LIN {X 0,Y 697.219,Z 878.166,A -85,B 0,C 180,E1 4075.669,E2 4075.669} C_VEL
LIN {X 0,Y 690.417,Z 859.31,A -85,B 0,C 180,E1 4076.202,E2 4076.202} C_VEL
LIN {X 0,Y 690.418,Z 859.31,A -85,B 0,C 180,E1 4081.164,E2 4081.164} C_VEL
LIN {X 0,Y 690.448,Z 859.31,A -85,B 0,C 180,E1 4086.339,E2 4086.339} C_VEL
LIN {X 0,Y 690.273,Z 859.31,A -85,B 0,C 180,E1 4091.743,E2 4091.743} C_VEL
LIN {X 0,Y 690.253,Z 859.31,A -85,B 0,C 180,E1 4097.131,E2 4097.131} C_VEL
LIN {X 0,Y 690.435,Z 859.31,A -85,B 0,C 180,E1 4102.194,E2 4102.194} C_VEL
LIN {X 0,Y 690.368,Z 859.31,A -85,B 0,C 180,E1 4106.732,E2 4106.732} C_VEL
LIN {X 0,Y 690.473,Z 859.31,A -85,B 0,C 180,E1 4112.567,E2 4112.567} C_VEL
LIN {X 0,Y 690.577,Z 859.31,A -85,B 0,C 180,E1 4117.159,E2 4117.159} C_VEL
LIN {X 0,Y 690.259,Z 859.31,A -85,B 0,C 180,E1 4122.108,E2 4122.108} C_VEL
LIN {X 0,Y 690.493,Z 859.31,A -85,B 0,C 180,E1 4127.328,E2 4127.328} C_VEL
LIN {X 0,Y 690.762,Z 859.31,A -85,B 0,C 180,E1 4132.441,E2 4132.441} C_VEL
LIN {X 0,Y 690.867,Z 859.31,A -85,B 0,C 180,E1 4137.488,E2 4137.488} C_VEL
LIN {X 0,Y 690.736,Z 859.31,A -85,B 0,C 180,E1 4142.516,E2 4142.516} C_VEL
LIN {X 0,Y 690.678,Z 859.31,A -85,B 0,C 180,E1 4146.298,E2 4146.298} C_VEL
LIN {X 0,Y 690.573,Z 859.31,A -85,B 0,C 180,E1 4151.388,E2 4151.388} C_VEL
LIN {X 0,Y 690.673,Z 859.31,A -85,B 0,C 180,E1 4156.569,E2 4156.569} C_VEL
LIN {X 0,Y 690.58,Z 859.31,A -85,B 0,C 180,E1 4158.902,E2 4158.902} C_VEL
LIN {X 0,Y 689.346,Z 859.31,A -85,B 0,C 180,E1 4159.621,E2 4159.621} C_VEL
LIN {X 0,Y 682.724,Z 859.31,A -85,B 0,C 180,E1 4161.574,E2 4161.574} C_VEL
LIN {X 0,Y 682.632,Z 859.31,A -85,B 0,C 180,E1 4161.759,E2 4161.759} C_VEL
LIN {X 0,Y 682.573,Z 859.31,A -85,B 0,C 180,E1 4166.353,E2 4166.353} C_VEL
LIN {X 0,Y 682.473,Z 859.31,A -85,B 0,C 180,E1 4170.701,E2 4170.701} C_VEL
LIN {X 0,Y 682.429,Z 859.31,A -85,B 0,C 180,E1 4175.253,E2 4175.253} C_VEL
LIN {X 0,Y 682.32,Z 859.31,A -85,B 0,C 180,E1 4180.082,E2 4180.082} C_VEL
LIN {X 0,Y 682.342,Z 859.31,A -85,B 0,C 180,E1 4185.273,E2 4185.273} C_VEL
LIN {X 0,Y 682.313,Z 859.31,A -85,B 0,C 180,E1 4189.906,E2 4189.906} C_VEL
LIN {X 0,Y 682.596,Z 859.31,A -85,B 0,C 180,E1 4195.202,E2 4195.202} C_VEL
LIN {X 0,Y 682.589,Z 859.31,A -85,B 0,C 180,E1 4196.549,E2 4196.549} C_VEL
LIN {X 0,Y 694.66,Z 886.241,A -85,B 0,C 180,E1 4197.535,E2 4197.535} C_VEL
LIN {X 0,Y 694.161,Z 942.115,A -85,B 0,C 180,E1 4198.336,E2 4198.336} C_VEL
LIN {X 0,Y 692.613,Z 987.576,A -85,B 0,C 180,E1 4199.516,E2 4199.516} C_VEL
LIN {X 0,Y 690.947,Z 1031.433,A -85,B 0,C 180,E1 4201.237,E2 4201.237} C_VEL
LIN {X 0,Y 689.086,Z 1070.916,A -85,B 0,C 180,E1 4203.334,E2 4203.334} C_VEL
LIN {X 0,Y 687.326,Z 1107.752,A -85,B 0,C 180,E1 4205.869,E2 4205.869} C_VEL
LIN {X 0,Y 685.7,Z 1142.826,A -85,B 0,C 180,E1 4208.975,E2 4208.975} C_VEL
LIN {X 0,Y 684.392,Z 1172.804,A -85,B 0,C 180,E1 4212.399,E2 4212.399} C_VEL
LIN {X 0,Y 683.648,Z 1196.132,A -85,B 0,C 180,E1 4215.888,E2 4215.888} C_VEL
LIN {X 0,Y 683.29,Z 1213.836,A -85,B 0,C 180,E1 4219.458,E2 4219.458} C_VEL
LIN {X 0,Y 683.115,Z 1226.068,A -85,B 0,C 180,E1 4222.992,E2 4222.992} C_VEL
LIN {X 0,Y 682.989,Z 1233.087,A -85,B 0,C 180,E1 4226.507,E2 4226.507} C_VEL
LIN {X 0,Y 683.008,Z 1235.5,A -85,B 0,C 180,E1 4230,E2 4230} C_VEL
LIN {X 0,Y 683.027,Z 1232.652,A -85,B 0,C 180,E1 4233.816,E2 4233.816} C_VEL
LIN {X 0,Y 683.081,Z 1226.069,A -85,B 0,C 180,E1 4237.008,E2 4237.008} C_VEL
LIN {X 0,Y 683.26,Z 1213.838,A -85,B 0,C 180,E1 4240.542,E2 4240.542} C_VEL
LIN {X 0,Y 683.653,Z 1196.132,A -85,B 0,C 180,E1 4244.111,E2 4244.111} C_VEL
LIN {X 0,Y 684.375,Z 1172.883,A -85,B 0,C 180,E1 4247.591,E2 4247.591} C_VEL
LIN {X 0,Y 685.586,Z 1144.349,A -85,B 0,C 180,E1 4250.869,E2 4250.869} C_VEL
LIN {X 0,Y 687.099,Z 1111.989,A -85,B 0,C 180,E1 4253.791,E2 4253.791} C_VEL
LIN {X 0,Y 688.909,Z 1076.012,A -85,B 0,C 180,E1 4256.35,E2 4256.35} C_VEL
LIN {X 0,Y 690.795,Z 1036.511,A -85,B 0,C 180,E1 4258.528,E2 4258.528} C_VEL
LIN {X 0,Y 692.579,Z 992.801,A -85,B 0,C 180,E1 4260.303,E2 4260.303} C_VEL
LIN {X 0,Y 693.916,Z 952.719,A -85,B 0,C 180,E1 4261.43,E2 4261.43} C_VEL
LIN {X 0,Y 694.73,Z 909.018,A -85,B 0,C 180,E1 4262.187,E2 4262.187} C_VEL
LIN {X 0,Y 694.325,Z 885.263,A -85,B 0,C 180,E1 4262.495,E2 4262.495} C_VEL
LIN {X 0,Y 682.567,Z 859.31,A -85,B 0,C 180,E1 4263.452,E2 4263.452} C_VEL
LIN {X 0,Y 682.392,Z 859.31,A -85,B 0,C 180,E1 4269.011,E2 4269.011} C_VEL
LIN {X 0,Y 682.579,Z 859.31,A -85,B 0,C 180,E1 4273.486,E2 4273.486} C_VEL
LIN {X 0,Y 682.368,Z 859.31,A -85,B 0,C 180,E1 4279.027,E2 4279.027} C_VEL
LIN {X 0,Y 682.363,Z 859.31,A -85,B 0,C 180,E1 4283.17,E2 4283.17} C_VEL
LIN {X 0,Y 682.444,Z 859.31,A -85,B 0,C 180,E1 4287.806,E2 4287.806} C_VEL
LIN {X 0,Y 682.632,Z 859.31,A -85,B 0,C 180,E1 4292.612,E2 4292.612} C_VEL
LIN {X 0,Y 682.664,Z 859.31,A -85,B 0,C 180,E1 4297.835,E2 4297.835} C_VEL
LIN {X 0,Y 682.691,Z 859.31,A -85,B 0,C 180,E1 4303.232,E2 4303.232} C_VEL
LIN {X 0,Y 682.688,Z 859.31,A -85,B 0,C 180,E1 4308.478,E2 4308.478} C_VEL
LIN {X 0,Y 682.896,Z 859.31,A -85,B 0,C 180,E1 4313.63,E2 4313.63} C_VEL
LIN {X 0,Y 682.841,Z 859.31,A -85,B 0,C 180,E1 4318.727,E2 4318.727} C_VEL
LIN {X 0,Y 682.863,Z 859.31,A -85,B 0,C 180,E1 4323.075,E2 4323.075} C_VEL
LIN {X 0,Y 682.774,Z 859.31,A -85,B 0,C 180,E1 4327.648,E2 4327.648} C_VEL
LIN {X 0,Y 682.771,Z 859.31,A -85,B 0,C 180,E1 4332.817,E2 4332.817} C_VEL
LIN {X 0,Y 682.691,Z 859.31,A -85,B 0,C 180,E1 4338.097,E2 4338.097} C_VEL
LIN {X 0,Y 682.561,Z 859.31,A -85,B 0,C 180,E1 4343.545,E2 4343.545} C_VEL
LIN {X 0,Y 682.547,Z 859.31,A -85,B 0,C 180,E1 4347.779,E2 4347.779} C_VEL
LIN {X 0,Y 682.439,Z 859.31,A -85,B 0,C 180,E1 4352.462,E2 4352.462} C_VEL
LIN {X 0,Y 682.458,Z 859.31,A -85,B 0,C 180,E1 4356.935,E2 4356.935} C_VEL
LIN {X 0,Y 682.378,Z 859.31,A -85,B 0,C 180,E1 4361.757,E2 4361.757} C_VEL
LIN {X 0,Y 682.362,Z 859.31,A -85,B 0,C 180,E1 4367.104,E2 4367.104} C_VEL
LIN {X 0,Y 682.426,Z 859.31,A -85,B 0,C 180,E1 4371.558,E2 4371.558} C_VEL
LIN {X 0,Y 682.493,Z 859.31,A -85,B 0,C 180,E1 4376.285,E2 4376.285} C_VEL
LIN {X 0,Y 682.432,Z 859.31,A -85,B 0,C 180,E1 4380.759,E2 4380.759} C_VEL
LIN {X 0,Y 682.609,Z 860.101,A -85,B 0,C 180,E1 4383.414,E2 4383.414} C_VEL
LIN {X 0,Y 690.644,Z 881.208,A -85,B 0,C 180,E1 4384.012,E2 4384.012} C_VEL
LIN {X 0,Y 690.138,Z 969.054,A -85,B 0,C 180,E1 4385.079,E2 4385.079} C_VEL
LIN {X 0,Y 689.243,Z 1008.749,A -85,B 0,C 180,E1 4386.059,E2 4386.059} C_VEL
LIN {X 0,Y 687.984,Z 1047.945,A -85,B 0,C 180,E1 4387.578,E2 4387.578} C_VEL
LIN {X 0,Y 686.6,Z 1083.977,A -85,B 0,C 180,E1 4389.557,E2 4389.557} C_VEL
LIN {X 0,Y 685.347,Z 1115.624,A -85,B 0,C 180,E1 4391.886,E2 4391.886} C_VEL
LIN {X 0,Y 684.434,Z 1141.565,A -85,B 0,C 180,E1 4394.374,E2 4394.374} C_VEL
LIN {X 0,Y 683.7,Z 1165.212,A -85,B 0,C 180,E1 4397.358,E2 4397.358} C_VEL
LIN {X 0,Y 683.315,Z 1182.757,A -85,B 0,C 180,E1 4400.374,E2 4400.374} C_VEL
LIN {X 0,Y 683.103,Z 1195.738,A -85,B 0,C 180,E1 4403.632,E2 4403.632} C_VEL
LIN {X 0,Y 683.082,Z 1202.285,A -85,B 0,C 180,E1 4406.328,E2 4406.328} C_VEL
LIN {X 0,Y 683.01,Z 1205.493,A -85,B 0,C 180,E1 4410,E2 4410} C_VEL
LIN {X 0,Y 683.084,Z 1203.836,A -85,B 0,C 180,E1 4412.543,E2 4412.543} C_VEL
LIN {X 0,Y 683.168,Z 1197.388,A -85,B 0,C 180,E1 4415.728,E2 4415.728} C_VEL
LIN {X 0,Y 683.254,Z 1185.646,A -85,B 0,C 180,E1 4418.931,E2 4418.931} C_VEL
LIN {X 0,Y 683.675,Z 1167.868,A -85,B 0,C 180,E1 4422.155,E2 4422.155} C_VEL
LIN {X 0,Y 684.244,Z 1145.639,A -85,B 0,C 180,E1 4425.083,E2 4425.083} C_VEL
LIN {X 0,Y 685.221,Z 1119.372,A -85,B 0,C 180,E1 4427.702,E2 4427.702} C_VEL
LIN {X 0,Y 686.442,Z 1088.334,A -85,B 0,C 180,E1 4430.068,E2 4430.068} C_VEL
LIN {X 0,Y 687.73,Z 1053.775,A -85,B 0,C 180,E1 4432.05,E2 4432.05} C_VEL
LIN {X 0,Y 688.945,Z 1018.152,A -85,B 0,C 180,E1 4433.536,E2 4433.536} C_VEL
LIN {X 0,Y 689.856,Z 981.67,A -85,B 0,C 180,E1 4434.576,E2 4434.576} C_VEL
LIN {X 0,Y 690.349,Z 943.118,A -85,B 0,C 180,E1 4435.21,E2 4435.21} C_VEL
LIN {X 0,Y 690.062,Z 880.068,A -85,B 0,C 180,E1 4435.934,E2 4435.934} C_VEL
LIN {X 0,Y 682.529,Z 859.31,A -85,B 0,C 180,E1 4436.555,E2 4436.555} C_VEL
LIN {X 0,Y 682.492,Z 859.31,A -85,B 0,C 180,E1 4442.199,E2 4442.199} C_VEL
LIN {X 0,Y 682.491,Z 859.31,A -85,B 0,C 180,E1 4446.961,E2 4446.961} C_VEL
LIN {X 0,Y 682.387,Z 859.31,A -85,B 0,C 180,E1 4451.773,E2 4451.773} C_VEL
LIN {X 0,Y 682.353,Z 859.31,A -85,B 0,C 180,E1 4457.124,E2 4457.124} C_VEL
LIN {X 0,Y 682.4,Z 859.31,A -85,B 0,C 180,E1 4461.57,E2 4461.57} C_VEL
LIN {X 0,Y 682.466,Z 859.31,A -85,B 0,C 180,E1 4466.296,E2 4466.296} C_VEL
LIN {X 0,Y 682.56,Z 859.31,A -85,B 0,C 180,E1 4472.222,E2 4472.222} C_VEL
LIN {X 0,Y 682.612,Z 859.31,A -85,B 0,C 180,E1 4476.457,E2 4476.457} C_VEL
LIN {X 0,Y 682.546,Z 859.31,A -85,B 0,C 180,E1 4480.556,E2 4480.556} C_VEL
LIN {X 0,Y 682.564,Z 859.31,A -85,B 0,C 180,E1 4485.871,E2 4485.871} C_VEL
LIN {X 0,Y 682.778,Z 859.31,A -85,B 0,C 180,E1 4491.067,E2 4491.067} C_VEL
LIN {X 0,Y 682.942,Z 859.31,A -85,B 0,C 180,E1 4496.186,E2 4496.186} C_VEL
LIN {X 0,Y 683.061,Z 859.31,A -85,B 0,C 180,E1 4501.273,E2 4501.273} C_VEL
LIN {X 0,Y 682.784,Z 859.31,A -85,B 0,C 180,E1 4506.371,E2 4506.371} C_VEL
LIN {X 0,Y 682.666,Z 859.31,A -85,B 0,C 180,E1 4511.522,E2 4511.522} C_VEL
LIN {X 0,Y 682.744,Z 859.31,A -85,B 0,C 180,E1 4516.767,E2 4516.767} C_VEL
LIN {X 0,Y 682.632,Z 859.31,A -85,B 0,C 180,E1 4521.759,E2 4521.759} C_VEL
LIN {X 0,Y 681.37,Z 859.31,A -85,B 0,C 180,E1 4522.485,E2 4522.485} C_VEL
LIN {X 0,Y 674.718,Z 859.31,A -85,B 0,C 180,E1 4524.458,E2 4524.458} C_VEL
LIN {X 0,Y 674.625,Z 859.31,A -85,B 0,C 180,E1 4524.645,E2 4524.645} C_VEL
LIN {X 0,Y 674.577,Z 859.31,A -85,B 0,C 180,E1 4529.609,E2 4529.609} C_VEL
LIN {X 0,Y 674.523,Z 859.31,A -85,B 0,C 180,E1 4534.159,E2 4534.159} C_VEL
LIN {X 0,Y 674.482,Z 859.31,A -85,B 0,C 180,E1 4538.97,E2 4538.97} C_VEL
LIN {X 0,Y 674.429,Z 859.31,A -85,B 0,C 180,E1 4544.135,E2 4544.135} C_VEL
LIN {X 0,Y 674.436,Z 859.31,A -85,B 0,C 180,E1 4549.794,E2 4549.794} C_VEL
LIN {X 0,Y 674.626,Z 859.31,A -85,B 0,C 180,E1 4554.268,E2 4554.268} C_VEL
LIN {X 0,Y 674.719,Z 860.083,A -85,B 0,C 180,E1 4556.128,E2 4556.128} C_VEL
LIN {X 0,Y 688.177,Z 890.762,A -85,B 0,C 180,E1 4557.246,E2 4557.246} C_VEL
LIN {X 0,Y 687.372,Z 943.616,A -85,B 0,C 180,E1 4558.022,E2 4558.022} C_VEL
LIN {X 0,Y 685.688,Z 989.724,A -85,B 0,C 180,E1 4559.246,E2 4559.246} C_VEL
LIN {X 0,Y 683.712,Z 1034.768,A -85,B 0,C 180,E1 4561.064,E2 4561.064} C_VEL
LIN {X 0,Y 681.56,Z 1076.167,A -85,B 0,C 180,E1 4563.354,E2 4563.354} C_VEL
LIN {X 0,Y 679.627,Z 1112.596,A -85,B 0,C 180,E1 4565.982,E2 4565.982} C_VEL
LIN {X 0,Y 678.016,Z 1144.493,A -85,B 0,C 180,E1 4568.902,E2 4568.902} C_VEL
LIN {X 0,Y 676.631,Z 1173.438,A -85,B 0,C 180,E1 4572.278,E2 4572.278} C_VEL
LIN {X 0,Y 675.848,Z 1196.131,A -85,B 0,C 180,E1 4575.722,E2 4575.722} C_VEL
LIN {X 0,Y 675.428,Z 1213.837,A -85,B 0,C 180,E1 4579.334,E2 4579.334} C_VEL
LIN {X 0,Y 675.218,Z 1226.068,A -85,B 0,C 180,E1 4582.91,E2 4582.91} C_VEL
LIN {X 0,Y 675.118,Z 1232.65,A -85,B 0,C 180,E1 4586.139,E2 4586.139} C_VEL
LIN {X 0,Y 675.137,Z 1235.5,A -85,B 0,C 180,E1 4590,E2 4590} C_VEL
LIN {X 0,Y 675.128,Z 1232.651,A -85,B 0,C 180,E1 4593.861,E2 4593.861} C_VEL
LIN {X 0,Y 675.18,Z 1226.069,A -85,B 0,C 180,E1 4597.09,E2 4597.09} C_VEL
LIN {X 0,Y 675.392,Z 1213.839,A -85,B 0,C 180,E1 4600.666,E2 4600.666} C_VEL
LIN {X 0,Y 675.851,Z 1196.13,A -85,B 0,C 180,E1 4604.278,E2 4604.278} C_VEL
LIN {X 0,Y 676.713,Z 1171.539,A -85,B 0,C 180,E1 4607.974,E2 4607.974} C_VEL
LIN {X 0,Y 678.114,Z 1141.776,A -85,B 0,C 180,E1 4611.384,E2 4611.384} C_VEL
LIN {X 0,Y 679.994,Z 1105.755,A -85,B 0,C 180,E1 4614.571,E2 4614.571} C_VEL
LIN {X 0,Y 682.155,Z 1066.242,A -85,B 0,C 180,E1 4617.259,E2 4617.259} C_VEL
LIN {X 0,Y 684.237,Z 1024.252,A -85,B 0,C 180,E1 4619.415,E2 4619.415} C_VEL
LIN {X 0,Y 686.078,Z 981.213,A -85,B 0,C 180,E1 4621.016,E2 4621.016} C_VEL
LIN {X 0,Y 687.436,Z 937.981,A -85,B 0,C 180,E1 4622.093,E2 4622.093} C_VEL
LIN {X 0,Y 687.755,Z 888.134,A -85,B 0,C 180,E1 4622.809,E2 4622.809} C_VEL
LIN {X 0,Y 674.633,Z 859.31,A -85,B 0,C 180,E1 4623.915,E2 4623.915} C_VEL
LIN {X 0,Y 674.513,Z 859.31,A -85,B 0,C 180,E1 4628.978,E2 4628.978} C_VEL
LIN {X 0,Y 674.668,Z 859.31,A -85,B 0,C 180,E1 4634.127,E2 4634.127} C_VEL
LIN {X 0,Y 674.487,Z 859.31,A -85,B 0,C 180,E1 4639.804,E2 4639.804} C_VEL
LIN {X 0,Y 674.432,Z 859.31,A -85,B 0,C 180,E1 4644.265,E2 4644.265} C_VEL
LIN {X 0,Y 674.542,Z 859.31,A -85,B 0,C 180,E1 4648.898,E2 4648.898} C_VEL
LIN {X 0,Y 674.702,Z 859.31,A -85,B 0,C 180,E1 4653.941,E2 4653.941} C_VEL
LIN {X 0,Y 674.735,Z 859.31,A -85,B 0,C 180,E1 4658.945,E2 4658.945} C_VEL
LIN {X 0,Y 674.764,Z 859.31,A -85,B 0,C 180,E1 4664.369,E2 4664.369} C_VEL
LIN {X 0,Y 674.856,Z 859.31,A -85,B 0,C 180,E1 4669.653,E2 4669.653} C_VEL
LIN {X 0,Y 674.899,Z 859.31,A -85,B 0,C 180,E1 4674.847,E2 4674.847} C_VEL
LIN {X 0,Y 675.011,Z 859.31,A -85,B 0,C 180,E1 4679.998,E2 4679.998} C_VEL
LIN {X 0,Y 675.106,Z 859.31,A -85,B 0,C 180,E1 4685.148,E2 4685.148} C_VEL
LIN {X 0,Y 674.799,Z 859.31,A -85,B 0,C 180,E1 4690.344,E2 4690.344} C_VEL
LIN {X 0,Y 674.786,Z 859.31,A -85,B 0,C 180,E1 4695.627,E2 4695.627} C_VEL
LIN {X 0,Y 674.731,Z 859.31,A -85,B 0,C 180,E1 4701.051,E2 4701.051} C_VEL
LIN {X 0,Y 674.634,Z 859.31,A -85,B 0,C 180,E1 4706.684,E2 4706.684} C_VEL
LIN {X 0,Y 674.525,Z 859.31,A -85,B 0,C 180,E1 4711.389,E2 4711.389} C_VEL
LIN {X 0,Y 674.494,Z 859.31,A -85,B 0,C 180,E1 4716.025,E2 4716.025} C_VEL
LIN {X 0,Y 674.449,Z 859.31,A -85,B 0,C 180,E1 4720.643,E2 4720.643} C_VEL
LIN {X 0,Y 674.414,Z 859.31,A -85,B 0,C 180,E1 4725.952,E2 4725.952} C_VEL
LIN {X 0,Y 674.504,Z 859.31,A -85,B 0,C 180,E1 4731.022,E2 4731.022} C_VEL
LIN {X 0,Y 674.589,Z 859.31,A -85,B 0,C 180,E1 4736.187,E2 4736.187} C_VEL
LIN {X 0,Y 674.546,Z 859.31,A -85,B 0,C 180,E1 4741.853,E2 4741.853} C_VEL
LIN {X 0,Y 674.64,Z 859.31,A -85,B 0,C 180,E1 4742.96,E2 4742.96} C_VEL
LIN {X 0,Y 683.587,Z 884.911,A -85,B 0,C 180,E1 4743.766,E2 4743.766} C_VEL
LIN {X 0,Y 682.976,Z 969.021,A -85,B 0,C 180,E1 4744.799,E2 4744.799} C_VEL
LIN {X 0,Y 681.97,Z 1009.288,A -85,B 0,C 180,E1 4745.805,E2 4745.805} C_VEL
LIN {X 0,Y 680.567,Z 1048.213,A -85,B 0,C 180,E1 4747.334,E2 4747.334} C_VEL
LIN {X 0,Y 679.069,Z 1084.367,A -85,B 0,C 180,E1 4749.347,E2 4749.347} C_VEL
LIN {X 0,Y 677.747,Z 1114.646,A -85,B 0,C 180,E1 4751.591,E2 4751.591} C_VEL
LIN {X 0,Y 676.664,Z 1142.43,A -85,B 0,C 180,E1 4754.288,E2 4754.288} C_VEL
LIN {X 0,Y 675.885,Z 1165.244,A -85,B 0,C 180,E1 4757.215,E2 4757.215} C_VEL
LIN {X 0,Y 675.442,Z 1183.007,A -85,B 0,C 180,E1 4760.314,E2 4760.314} C_VEL
LIN {X 0,Y 675.214,Z 1195.736,A -85,B 0,C 180,E1 4763.558,E2 4763.558} C_VEL
LIN {X 0,Y 675.205,Z 1202.016,A -85,B 0,C 180,E1 4766.14,E2 4766.14} C_VEL
LIN {X 0,Y 675.121,Z 1205.119,A -85,B 0,C 180,E1 4768.714,E2 4768.714} C_VEL
LIN {X 0,Y 675.219,Z 1205.047,A -85,B 0,C 180,E1 4771.286,E2 4771.286} C_VEL
LIN {X 0,Y 675.246,Z 1200.619,A -85,B 0,C 180,E1 4774.505,E2 4774.505} C_VEL
LIN {X 0,Y 675.389,Z 1189.741,A -85,B 0,C 180,E1 4778.061,E2 4778.061} C_VEL
LIN {X 0,Y 675.739,Z 1173.885,A -85,B 0,C 180,E1 4781.316,E2 4781.316} C_VEL
LIN {X 0,Y 676.263,Z 1153.81,A -85,B 0,C 180,E1 4784.269,E2 4784.269} C_VEL
LIN {X 0,Y 677.194,Z 1128.422,A -85,B 0,C 180,E1 4787.074,E2 4787.074} C_VEL
LIN {X 0,Y 678.461,Z 1098.701,A -85,B 0,C 180,E1 4789.574,E2 4789.574} C_VEL
LIN {X 0,Y 679.837,Z 1065.972,A -85,B 0,C 180,E1 4791.664,E2 4791.664} C_VEL
LIN {X 0,Y 681.195,Z 1030.24,A -85,B 0,C 180,E1 4793.352,E2 4793.352} C_VEL
LIN {X 0,Y 682.38,Z 992.126,A -85,B 0,C 180,E1 4794.599,E2 4794.599} C_VEL
LIN {X 0,Y 683.139,Z 953.244,A -85,B 0,C 180,E1 4795.364,E2 4795.364} C_VEL
LIN {X 0,Y 682.79,Z 881.512,A -85,B 0,C 180,E1 4796.227,E2 4796.227} C_VEL
LIN {X 0,Y 674.627,Z 859.31,A -85,B 0,C 180,E1 4796.981,E2 4796.981} C_VEL
LIN {X 0,Y 674.596,Z 859.31,A -85,B 0,C 180,E1 4802.622,E2 4802.622} C_VEL
LIN {X 0,Y 674.525,Z 859.31,A -85,B 0,C 180,E1 4808.185,E2 4808.185} C_VEL
LIN {X 0,Y 674.459,Z 859.31,A -85,B 0,C 180,E1 4812.377,E2 4812.377} C_VEL
LIN {X 0,Y 674.454,Z 859.31,A -85,B 0,C 180,E1 4817.852,E2 4817.852} C_VEL
LIN {X 0,Y 674.537,Z 859.31,A -85,B 0,C 180,E1 4822.675,E2 4822.675} C_VEL
LIN {X 0,Y 674.511,Z 859.31,A -85,B 0,C 180,E1 4827.385,E2 4827.385} C_VEL
LIN {X 0,Y 674.595,Z 859.31,A -85,B 0,C 180,E1 4831.865,E2 4831.865} C_VEL
LIN {X 0,Y 674.674,Z 859.31,A -85,B 0,C 180,E1 4837.05,E2 4837.05} C_VEL
LIN {X 0,Y 674.466,Z 859.31,A -85,B 0,C 180,E1 4841.674,E2 4841.674} C_VEL
LIN {X 0,Y 674.654,Z 859.31,A -85,B 0,C 180,E1 4847.026,E2 4847.026} C_VEL
LIN {X 0,Y 674.941,Z 859.31,A -85,B 0,C 180,E1 4852.262,E2 4852.262} C_VEL
LIN {X 0,Y 675.075,Z 859.31,A -85,B 0,C 180,E1 4857.429,E2 4857.429} C_VEL
LIN {X 0,Y 674.956,Z 859.31,A -85,B 0,C 180,E1 4862.575,E2 4862.575} C_VEL
LIN {X 0,Y 674.874,Z 859.31,A -85,B 0,C 180,E1 4866.446,E2 4866.446} C_VEL
LIN {X 0,Y 674.788,Z 859.31,A -85,B 0,C 180,E1 4870.348,E2 4870.348} C_VEL
LIN {X 0,Y 674.799,Z 859.31,A -85,B 0,C 180,E1 4875.63,E2 4875.63} C_VEL
LIN {X 0,Y 674.785,Z 859.31,A -85,B 0,C 180,E1 4881.053,E2 4881.053} C_VEL
LIN {X 0,Y 674.625,Z 859.31,A -85,B 0,C 180,E1 4884.645,E2 4884.645} C_VEL
LIN {X 0,Y 670.662,Z 859.31,A -85,B 0,C 180,E1 4886.09,E2 4886.09} C_VEL
LIN {X 0,Y 666.704,Z 859.31,A -85,B 0,C 180,E1 4887.552,E2 4887.552} C_VEL
LIN {X 0,Y 666.618,Z 859.31,A -85,B 0,C 180,E1 4893.054,E2 4893.054} C_VEL
LIN {X 0,Y 666.601,Z 859.31,A -85,B 0,C 180,E1 4897.852,E2 4897.852} C_VEL
LIN {X 0,Y 666.477,Z 859.31,A -85,B 0,C 180,E1 4903.319,E2 4903.319} C_VEL
LIN {X 0,Y 666.481,Z 859.31,A -85,B 0,C 180,E1 4908.75,E2 4908.75} C_VEL
LIN {X 0,Y 666.685,Z 859.31,A -85,B 0,C 180,E1 4913.775,E2 4913.775} C_VEL
LIN {X 0,Y 666.773,Z 859.31,A -85,B 0,C 180,E1 4915.739,E2 4915.739} C_VEL
LIN {X 0,Y 676.305,Z 880.508,A -85,B 0,C 180,E1 4916.468,E2 4916.468} C_VEL
LIN {X 0,Y 681.457,Z 891.656,A -85,B 0,C 180,E1 4916.892,E2 4916.892} C_VEL
LIN {X 0,Y 680.649,Z 943.593,A -85,B 0,C 180,E1 4917.667,E2 4917.667} C_VEL
LIN {X 0,Y 678.842,Z 989.466,A -85,B 0,C 180,E1 4918.893,E2 4918.893} C_VEL
LIN {X 0,Y 676.675,Z 1035.331,A -85,B 0,C 180,E1 4920.761,E2 4920.761} C_VEL
LIN {X 0,Y 674.296,Z 1076.831,A -85,B 0,C 180,E1 4923.087,E2 4923.087} C_VEL
LIN {X 0,Y 672.129,Z 1113.665,A -85,B 0,C 180,E1 4925.787,E2 4925.787} C_VEL
LIN {X 0,Y 670.365,Z 1145.862,A -85,B 0,C 180,E1 4928.797,E2 4928.797} C_VEL
LIN {X 0,Y 668.912,Z 1173.914,A -85,B 0,C 180,E1 4932.133,E2 4932.133} C_VEL
LIN {X 0,Y 668.036,Z 1196.13,A -85,B 0,C 180,E1 4935.551,E2 4935.551} C_VEL
LIN {X 0,Y 667.568,Z 1213.837,A -85,B 0,C 180,E1 4939.207,E2 4939.207} C_VEL
LIN {X 0,Y 667.325,Z 1226.068,A -85,B 0,C 180,E1 4942.826,E2 4942.826} C_VEL
LIN {X 0,Y 667.224,Z 1232.65,A -85,B 0,C 180,E1 4946.093,E2 4946.093} C_VEL
LIN {X 0,Y 667.237,Z 1235.5,A -85,B 0,C 180,E1 4950,E2 4950} C_VEL
LIN {X 0,Y 667.231,Z 1232.651,A -85,B 0,C 180,E1 4953.906,E2 4953.906} C_VEL
LIN {X 0,Y 667.284,Z 1226.069,A -85,B 0,C 180,E1 4957.175,E2 4957.175} C_VEL
LIN {X 0,Y 667.528,Z 1213.84,A -85,B 0,C 180,E1 4960.794,E2 4960.794} C_VEL
LIN {X 0,Y 668.037,Z 1196.129,A -85,B 0,C 180,E1 4964.448,E2 4964.448} C_VEL
LIN {X 0,Y 669.015,Z 1171.677,A -85,B 0,C 180,E1 4968.17,E2 4968.17} C_VEL
LIN {X 0,Y 670.587,Z 1141.188,A -85,B 0,C 180,E1 4971.696,E2 4971.696} C_VEL
LIN {X 0,Y 672.667,Z 1105.263,A -85,B 0,C 180,E1 4974.895,E2 4974.895} C_VEL
LIN {X 0,Y 674.957,Z 1066.239,A -85,B 0,C 180,E1 4977.574,E2 4977.574} C_VEL
LIN {X 0,Y 677.288,Z 1023.55,A -85,B 0,C 180,E1 4979.781,E2 4979.781} C_VEL
LIN {X 0,Y 679.279,Z 980.059,A -85,B 0,C 180,E1 4981.399,E2 4981.399} C_VEL
LIN {X 0,Y 680.782,Z 935.996,A -85,B 0,C 180,E1 4982.483,E2 4982.483} C_VEL
LIN {X 0,Y 680.982,Z 890.343,A -85,B 0,C 180,E1 4983.15,E2 4983.15} C_VEL
LIN {X 0,Y 666.851,Z 860.732,A -85,B 0,C 180,E1 4984.225,E2 4984.225} C_VEL
LIN {X 0,Y 666.711,Z 859.31,A -85,B 0,C 180,E1 4984.302,E2 4984.302} C_VEL
LIN {X 0,Y 666.57,Z 859.31,A -85,B 0,C 180,E1 4989.532,E2 4989.532} C_VEL
LIN {X 0,Y 666.662,Z 859.31,A -85,B 0,C 180,E1 4994.798,E2 4994.798} C_VEL
LIN {X 0,Y 666.567,Z 859.31,A -85,B 0,C 180,E1 5000.616,E2 5000.616} C_VEL
LIN {X 0,Y 666.52,Z 859.31,A -85,B 0,C 180,E1 5005.372,E2 5005.372} C_VEL
LIN {X 0,Y 666.624,Z 859.31,A -85,B 0,C 180,E1 5010.002,E2 5010.002} C_VEL
LIN {X 0,Y 666.768,Z 859.31,A -85,B 0,C 180,E1 5015.372,E2 5015.372} C_VEL
LIN {X 0,Y 666.803,Z 859.31,A -85,B 0,C 180,E1 5020.074,E2 5020.074} C_VEL
LIN {X 0,Y 666.845,Z 859.31,A -85,B 0,C 180,E1 5024.179,E2 5024.179} C_VEL
LIN {X 0,Y 666.932,Z 859.31,A -85,B 0,C 180,E1 5029.529,E2 5029.529} C_VEL
LIN {X 0,Y 667.009,Z 859.31,A -85,B 0,C 180,E1 5034.786,E2 5034.786} C_VEL
LIN {X 0,Y 667.074,Z 859.31,A -85,B 0,C 180,E1 5038.697,E2 5038.697} C_VEL
LIN {X 0,Y 667.07,Z 859.31,A -85,B 0,C 180,E1 5042.601,E2 5042.601} C_VEL
LIN {X 0,Y 666.962,Z 859.31,A -85,B 0,C 180,E1 5046.519,E2 5046.519} C_VEL
LIN {X 0,Y 666.896,Z 859.31,A -85,B 0,C 180,E1 5051.795,E2 5051.795} C_VEL
LIN {X 0,Y 666.854,Z 859.31,A -85,B 0,C 180,E1 5057.377,E2 5057.377} C_VEL
LIN {X 0,Y 666.728,Z 859.31,A -85,B 0,C 180,E1 5062.72,E2 5062.72} C_VEL
LIN {X 0,Y 666.669,Z 859.31,A -85,B 0,C 180,E1 5067.571,E2 5067.571} C_VEL
LIN {X 0,Y 666.615,Z 859.31,A -85,B 0,C 180,E1 5073.05,E2 5073.05} C_VEL
LIN {X 0,Y 666.606,Z 859.31,A -85,B 0,C 180,E1 5077.847,E2 5077.847} C_VEL
LIN {X 0,Y 666.468,Z 859.31,A -85,B 0,C 180,E1 5083.318,E2 5083.318} C_VEL
LIN {X 0,Y 666.494,Z 859.31,A -85,B 0,C 180,E1 5088.752,E2 5088.752} C_VEL
LIN {X 0,Y 666.661,Z 859.31,A -85,B 0,C 180,E1 5093.774,E2 5093.774} C_VEL
LIN {X 0,Y 666.596,Z 859.31,A -85,B 0,C 180,E1 5098.478,E2 5098.478} C_VEL
LIN {X 0,Y 666.724,Z 859.31,A -85,B 0,C 180,E1 5102.531,E2 5102.531} C_VEL
LIN {X 0,Y 676.777,Z 885.125,A -85,B 0,C 180,E1 5103.408,E2 5103.408} C_VEL
LIN {X 0,Y 675.999,Z 968.354,A -85,B 0,C 180,E1 5104.475,E2 5104.475} C_VEL
LIN {X 0,Y 674.765,Z 1007.317,A -85,B 0,C 180,E1 5105.469,E2 5105.469} C_VEL
LIN {X 0,Y 673.291,Z 1046.299,A -85,B 0,C 180,E1 5106.982,E2 5106.982} C_VEL
LIN {X 0,Y 671.684,Z 1082.811,A -85,B 0,C 180,E1 5109.004,E2 5109.004} C_VEL
LIN {X 0,Y 670.124,Z 1114.638,A -85,B 0,C 180,E1 5111.374,E2 5111.374} C_VEL
LIN {X 0,Y 668.907,Z 1142.424,A -85,B 0,C 180,E1 5114.101,E2 5114.101} C_VEL
LIN {X 0,Y 668.123,Z 1164.113,A -85,B 0,C 180,E1 5116.892,E2 5116.892} C_VEL
LIN {X 0,Y 667.624,Z 1181.463,A -85,B 0,C 180,E1 5119.869,E2 5119.869} C_VEL
LIN {X 0,Y 667.391,Z 1194.77,A -85,B 0,C 180,E1 5123.154,E2 5123.154} C_VEL
LIN {X 0,Y 667.311,Z 1202.016,A -85,B 0,C 180,E1 5126.094,E2 5126.094} C_VEL
LIN {X 0,Y 667.221,Z 1205.119,A -85,B 0,C 180,E1 5128.699,E2 5128.699} C_VEL
LIN {X 0,Y 667.317,Z 1205.047,A -85,B 0,C 180,E1 5131.301,E2 5131.301} C_VEL
LIN {X 0,Y 667.361,Z 1200.621,A -85,B 0,C 180,E1 5134.558,E2 5134.558} C_VEL
LIN {X 0,Y 667.518,Z 1189.743,A -85,B 0,C 180,E1 5138.157,E2 5138.157} C_VEL
LIN {X 0,Y 667.901,Z 1173.887,A -85,B 0,C 180,E1 5141.45,E2 5141.45} C_VEL
LIN {X 0,Y 668.474,Z 1153.813,A -85,B 0,C 180,E1 5144.439,E2 5144.439} C_VEL
LIN {X 0,Y 669.493,Z 1128.631,A -85,B 0,C 180,E1 5147.257,E2 5147.257} C_VEL
LIN {X 0,Y 670.883,Z 1098.706,A -85,B 0,C 180,E1 5149.804,E2 5149.804} C_VEL
LIN {X 0,Y 672.424,Z 1065.979,A -85,B 0,C 180,E1 5151.915,E2 5151.915} C_VEL
LIN {X 0,Y 673.932,Z 1029.418,A -85,B 0,C 180,E1 5153.654,E2 5153.654} C_VEL
LIN {X 0,Y 675.356,Z 990.18,A -85,B 0,C 180,E1 5154.939,E2 5154.939} C_VEL
LIN {X 0,Y 676.221,Z 953.656,A -85,B 0,C 180,E1 5155.681,E2 5155.681} C_VEL
LIN {X 0,Y 676.308,Z 884.254,A -85,B 0,C 180,E1 5156.536,E2 5156.536} C_VEL
LIN {X 0,Y 666.712,Z 859.31,A -85,B 0,C 180,E1 5157.403,E2 5157.403} C_VEL
LIN {X 0,Y 666.678,Z 859.31,A -85,B 0,C 180,E1 5163.059,E2 5163.059} C_VEL
LIN {X 0,Y 666.632,Z 859.31,A -85,B 0,C 180,E1 5167.86,E2 5167.86} C_VEL
LIN {X 0,Y 666.46,Z 859.31,A -85,B 0,C 180,E1 5173.336,E2 5173.336} C_VEL
LIN {X 0,Y 666.486,Z 859.31,A -85,B 0,C 180,E1 5178.767,E2 5178.767} C_VEL
LIN {X 0,Y 666.662,Z 859.31,A -85,B 0,C 180,E1 5183.788,E2 5183.788} C_VEL
LIN {X 0,Y 666.574,Z 859.31,A -85,B 0,C 180,E1 5188.488,E2 5188.488} C_VEL
LIN {X 0,Y 666.706,Z 859.31,A -85,B 0,C 180,E1 5192.973,E2 5192.973} C_VEL
LIN {X 0,Y 666.779,Z 859.31,A -85,B 0,C 180,E1 5197.282,E2 5197.282} C_VEL
LIN {X 0,Y 666.586,Z 859.31,A -85,B 0,C 180,E1 5201.45,E2 5201.45} C_VEL
LIN {X 0,Y 666.751,Z 859.31,A -85,B 0,C 180,E1 5206.869,E2 5206.869} C_VEL
LIN {X 0,Y 667.027,Z 859.31,A -85,B 0,C 180,E1 5212.17,E2 5212.17} C_VEL
LIN {X 0,Y 667.197,Z 859.31,A -85,B 0,C 180,E1 5217.399,E2 5217.399} C_VEL
LIN {X 0,Y 667.069,Z 859.31,A -85,B 0,C 180,E1 5222.605,E2 5222.605} C_VEL
LIN {X 0,Y 666.965,Z 859.31,A -85,B 0,C 180,E1 5226.523,E2 5226.523} C_VEL
LIN {X 0,Y 666.856,Z 859.31,A -85,B 0,C 180,E1 5231.799,E2 5231.799} C_VEL
LIN {X 0,Y 666.881,Z 859.31,A -85,B 0,C 180,E1 5237.383,E2 5237.383} C_VEL
LIN {X 0,Y 666.791,Z 859.31,A -85,B 0,C 180,E1 5242.722,E2 5242.722} C_VEL
LIN {X 0,Y 666.704,Z 859.31,A -85,B 0,C 180,E1 5247.552,E2 5247.552} C_VEL
LIN {X 0,Y 665.467,Z 859.31,A -85,B 0,C 180,E1 5248.295,E2 5248.295} C_VEL
LIN {X 0,Y 658.829,Z 859.31,A -85,B 0,C 180,E1 5250.312,E2 5250.312} C_VEL
LIN {X 0,Y 658.718,Z 859.31,A -85,B 0,C 180,E1 5250.503,E2 5250.503} C_VEL
LIN {X 0,Y 658.68,Z 859.31,A -85,B 0,C 180,E1 5255.1,E2 5255.1} C_VEL
LIN {X 0,Y 658.537,Z 859.31,A -85,B 0,C 180,E1 5260.595,E2 5260.595} C_VEL
LIN {X 0,Y 658.519,Z 859.31,A -85,B 0,C 180,E1 5265.493,E2 5265.493} C_VEL
LIN {X 0,Y 658.553,Z 859.31,A -85,B 0,C 180,E1 5269.889,E2 5269.889} C_VEL
LIN {X 0,Y 658.812,Z 859.31,A -85,B 0,C 180,E1 5275.359,E2 5275.359} C_VEL
LIN {X 0,Y 668.893,Z 881.832,A -85,B 0,C 180,E1 5276.12,E2 5276.12} C_VEL
LIN {X 0,Y 674.712,Z 893.747,A -85,B 0,C 180,E1 5276.544,E2 5276.544} C_VEL
LIN {X 0,Y 673.897,Z 945.115,A -85,B 0,C 180,E1 5277.34,E2 5277.34} C_VEL
LIN {X 0,Y 671.97,Z 990.38,A -85,B 0,C 180,E1 5278.571,E2 5278.571} C_VEL
LIN {X 0,Y 669.679,Z 1035.455,A -85,B 0,C 180,E1 5280.432,E2 5280.432} C_VEL
LIN {X 0,Y 667.089,Z 1077.091,A -85,B 0,C 180,E1 5282.789,E2 5282.789} C_VEL
LIN {X 0,Y 664.718,Z 1113.736,A -85,B 0,C 180,E1 5285.505,E2 5285.505} C_VEL
LIN {X 0,Y 662.784,Z 1145.86,A -85,B 0,C 180,E1 5288.543,E2 5288.543} C_VEL
LIN {X 0,Y 661.193,Z 1173.916,A -85,B 0,C 180,E1 5291.917,E2 5291.917} C_VEL
LIN {X 0,Y 660.237,Z 1196.128,A -85,B 0,C 180,E1 5295.377,E2 5295.377} C_VEL
LIN {X 0,Y 659.706,Z 1213.838,A -85,B 0,C 180,E1 5299.076,E2 5299.076} C_VEL
LIN {X 0,Y 659.435,Z 1226.068,A -85,B 0,C 180,E1 5302.739,E2 5302.739} C_VEL
LIN {X 0,Y 659.326,Z 1232.649,A -85,B 0,C 180,E1 5306.046,E2 5306.046} C_VEL
LIN {X 0,Y 659.343,Z 1235.5,A -85,B 0,C 180,E1 5310,E2 5310} C_VEL
LIN {X 0,Y 659.333,Z 1232.651,A -85,B 0,C 180,E1 5313.953,E2 5313.953} C_VEL
LIN {X 0,Y 659.392,Z 1226.069,A -85,B 0,C 180,E1 5317.261,E2 5317.261} C_VEL
LIN {X 0,Y 659.667,Z 1213.84,A -85,B 0,C 180,E1 5320.924,E2 5320.924} C_VEL
LIN {X 0,Y 660.239,Z 1196.127,A -85,B 0,C 180,E1 5324.623,E2 5324.623} C_VEL
LIN {X 0,Y 661.306,Z 1171.673,A -85,B 0,C 180,E1 5328.39,E2 5328.39} C_VEL
LIN {X 0,Y 662.979,Z 1141.804,A -85,B 0,C 180,E1 5331.894,E2 5331.894} C_VEL
LIN {X 0,Y 665.215,Z 1106.38,A -85,B 0,C 180,E1 5335.104,E2 5335.104} C_VEL
LIN {X 0,Y 667.767,Z 1066.444,A -85,B 0,C 180,E1 5337.883,E2 5337.883} C_VEL
LIN {X 0,Y 670.238,Z 1024.936,A -85,B 0,C 180,E1 5340.058,E2 5340.058} C_VEL
LIN {X 0,Y 672.384,Z 982.623,A -85,B 0,C 180,E1 5341.672,E2 5341.672} C_VEL
LIN {X 0,Y 674.039,Z 938.784,A -85,B 0,C 180,E1 5342.794,E2 5342.794} C_VEL
LIN {X 0,Y 674.254,Z 892.584,A -85,B 0,C 180,E1 5343.496,E2 5343.496} C_VEL
LIN {X 0,Y 658.925,Z 860.75,A -85,B 0,C 180,E1 5344.595,E2 5344.595} C_VEL
LIN {X 0,Y 658.761,Z 859.31,A -85,B 0,C 180,E1 5344.64,E2 5344.64} C_VEL
LIN {X 0,Y 658.611,Z 859.31,A -85,B 0,C 180,E1 5350.106,E2 5350.106} C_VEL
LIN {X 0,Y 658.709,Z 859.31,A -85,B 0,C 180,E1 5355.489,E2 5355.489} C_VEL
LIN {X 0,Y 658.586,Z 859.31,A -85,B 0,C 180,E1 5359.902,E2 5359.902} C_VEL
LIN {X 0,Y 658.621,Z 859.31,A -85,B 0,C 180,E1 5364.897,E2 5364.897} C_VEL
LIN {X 0,Y 658.738,Z 859.31,A -85,B 0,C 180,E1 5369.605,E2 5369.605} C_VEL
LIN {X 0,Y 658.845,Z 859.31,A -85,B 0,C 180,E1 5374.094,E2 5374.094} C_VEL
LIN {X 0,Y 658.888,Z 859.31,A -85,B 0,C 180,E1 5378.414,E2 5378.414} C_VEL
LIN {X 0,Y 658.933,Z 859.31,A -85,B 0,C 180,E1 5383.984,E2 5383.984} C_VEL
LIN {X 0,Y 659.007,Z 859.31,A -85,B 0,C 180,E1 5389.401,E2 5389.401} C_VEL
LIN {X 0,Y 659.105,Z 859.31,A -85,B 0,C 180,E1 5394.723,E2 5394.723} C_VEL
LIN {X 0,Y 659.198,Z 859.31,A -85,B 0,C 180,E1 5398.681,E2 5398.681} C_VEL
LIN {X 0,Y 659.168,Z 859.31,A -85,B 0,C 180,E1 5402.633,E2 5402.633} C_VEL
LIN {X 0,Y 659.053,Z 859.31,A -85,B 0,C 180,E1 5406.598,E2 5406.598} C_VEL
LIN {X 0,Y 659.019,Z 859.31,A -85,B 0,C 180,E1 5411.938,E2 5411.938} C_VEL
LIN {X 0,Y 658.959,Z 859.31,A -85,B 0,C 180,E1 5417.387,E2 5417.387} C_VEL
LIN {X 0,Y 658.843,Z 859.31,A -85,B 0,C 180,E1 5421.584,E2 5421.584} C_VEL
LIN {X 0,Y 658.777,Z 859.31,A -85,B 0,C 180,E1 5426.226,E2 5426.226} C_VEL
LIN {X 0,Y 658.732,Z 859.31,A -85,B 0,C 180,E1 5431.667,E2 5431.667} C_VEL
LIN {X 0,Y 658.693,Z 859.31,A -85,B 0,C 180,E1 5436.722,E2 5436.722} C_VEL
LIN {X 0,Y 658.561,Z 859.31,A -85,B 0,C 180,E1 5441.84,E2 5441.84} C_VEL
LIN {X 0,Y 658.53,Z 859.31,A -85,B 0,C 180,E1 5447.4,E2 5447.4} C_VEL
LIN {X 0,Y 658.652,Z 859.31,A -85,B 0,C 180,E1 5451.599,E2 5451.599} C_VEL
LIN {X 0,Y 658.702,Z 859.31,A -85,B 0,C 180,E1 5456.489,E2 5456.489} C_VEL
LIN {X 0,Y 658.772,Z 859.596,A -85,B 0,C 180,E1 5462.093,E2 5462.093} C_VEL
LIN {X 0,Y 670.192,Z 888.549,A -85,B 0,C 180,E1 5463.091,E2 5463.091} C_VEL
LIN {X 0,Y 669.269,Z 968.718,A -85,B 0,C 180,E1 5464.125,E2 5464.125} C_VEL
LIN {X 0,Y 667.913,Z 1007.259,A -85,B 0,C 180,E1 5465.122,E2 5465.122} C_VEL
LIN {X 0,Y 666.082,Z 1044.758,A -85,B 0,C 180,E1 5466.629,E2 5466.629} C_VEL
LIN {X 0,Y 664.244,Z 1082.27,A -85,B 0,C 180,E1 5468.721,E2 5468.721} C_VEL
LIN {X 0,Y 662.527,Z 1114.63,A -85,B 0,C 180,E1 5471.152,E2 5471.152} C_VEL
LIN {X 0,Y 661.196,Z 1142.04,A -85,B 0,C 180,E1 5473.867,E2 5473.867} C_VEL
LIN {X 0,Y 660.338,Z 1164.11,A -85,B 0,C 180,E1 5476.734,E2 5476.734} C_VEL
LIN {X 0,Y 659.783,Z 1181.461,A -85,B 0,C 180,E1 5479.747,E2 5479.747} C_VEL
LIN {X 0,Y 659.505,Z 1194.768,A -85,B 0,C 180,E1 5483.072,E2 5483.072} C_VEL
LIN {X 0,Y 659.413,Z 1202.014,A -85,B 0,C 180,E1 5486.047,E2 5486.047} C_VEL
LIN {X 0,Y 659.333,Z 1205.119,A -85,B 0,C 180,E1 5488.683,E2 5488.683} C_VEL
LIN {X 0,Y 659.423,Z 1205.048,A -85,B 0,C 180,E1 5491.317,E2 5491.317} C_VEL
LIN {X 0,Y 659.474,Z 1200.622,A -85,B 0,C 180,E1 5494.613,E2 5494.613} C_VEL
LIN {X 0,Y 659.639,Z 1189.914,A -85,B 0,C 180,E1 5498.213,E2 5498.213} C_VEL
LIN {X 0,Y 660.081,Z 1173.89,A -85,B 0,C 180,E1 5501.588,E2 5501.588} C_VEL
LIN {X 0,Y 660.714,Z 1152.691,A -85,B 0,C 180,E1 5504.756,E2 5504.756} C_VEL
LIN {X 0,Y 661.863,Z 1127.503,A -85,B 0,C 180,E1 5507.573,E2 5507.573} C_VEL
LIN {X 0,Y 663.389,Z 1097.667,A -85,B 0,C 180,E1 5510.116,E2 5510.116} C_VEL
LIN {X 0,Y 665.099,Z 1064.587,A -85,B 0,C 180,E1 5512.25,E2 5512.25} C_VEL
LIN {X 0,Y 667.011,Z 1026.339,A -85,B 0,C 180,E1 5514.092,E2 5514.092} C_VEL
LIN {X 0,Y 668.638,Z 988.633,A -85,B 0,C 180,E1 5515.334,E2 5515.334} C_VEL
LIN {X 0,Y 669.588,Z 950.055,A -85,B 0,C 180,E1 5516.088,E2 5516.088} C_VEL
LIN {X 0,Y 669.447,Z 885.862,A -85,B 0,C 180,E1 5516.891,E2 5516.891} C_VEL
LIN {X 0,Y 658.75,Z 859.31,A -85,B 0,C 180,E1 5517.88,E2 5517.88} C_VEL
LIN {X 0,Y 658.713,Z 859.31,A -85,B 0,C 180,E1 5523.511,E2 5523.511} C_VEL
LIN {X 0,Y 658.654,Z 859.31,A -85,B 0,C 180,E1 5528.56,E2 5528.56} C_VEL
LIN {X 0,Y 658.519,Z 859.31,A -85,B 0,C 180,E1 5533.656,E2 5533.656} C_VEL
LIN {X 0,Y 658.548,Z 859.31,A -85,B 0,C 180,E1 5538.159,E2 5538.159} C_VEL
LIN {X 0,Y 658.759,Z 859.31,A -85,B 0,C 180,E1 5543.618,E2 5543.618} C_VEL
LIN {X 0,Y 658.688,Z 859.31,A -85,B 0,C 180,E1 5548.34,E2 5548.34} C_VEL
LIN {X 0,Y 658.804,Z 859.31,A -85,B 0,C 180,E1 5554.096,E2 5554.096} C_VEL
LIN {X 0,Y 658.872,Z 859.31,A -85,B 0,C 180,E1 5558.417,E2 5558.417} C_VEL
LIN {X 0,Y 658.709,Z 859.31,A -85,B 0,C 180,E1 5563.982,E2 5563.982} C_VEL
LIN {X 0,Y 659.044,Z 859.31,A -85,B 0,C 180,E1 5569.405,E2 5569.405} C_VEL
LIN {X 0,Y 659.118,Z 859.31,A -85,B 0,C 180,E1 5574.727,E2 5574.727} C_VEL
LIN {X 0,Y 659.201,Z 859.31,A -85,B 0,C 180,E1 5578.685,E2 5578.685} C_VEL
LIN {X 0,Y 659.167,Z 859.31,A -85,B 0,C 180,E1 5582.636,E2 5582.636} C_VEL
LIN {X 0,Y 659.055,Z 859.31,A -85,B 0,C 180,E1 5586.601,E2 5586.601} C_VEL
LIN {X 0,Y 658.96,Z 859.31,A -85,B 0,C 180,E1 5591.943,E2 5591.943} C_VEL
LIN {X 0,Y 658.986,Z 859.31,A -85,B 0,C 180,E1 5597.39,E2 5597.39} C_VEL
LIN {X 0,Y 658.908,Z 859.31,A -85,B 0,C 180,E1 5601.585,E2 5601.585} C_VEL
LIN {X 0,Y 658.806,Z 859.31,A -85,B 0,C 180,E1 5606.23,E2 5606.23} C_VEL
LIN {X 0,Y 658.718,Z 859.31,A -85,B 0,C 180,E1 5610.503,E2 5610.503} C_VEL
LIN {X 0,Y 654.663,Z 859.31,A -85,B 0,C 180,E1 5611.992,E2 5611.992} C_VEL
LIN {X 0,Y 650.712,Z 859.31,A -85,B 0,C 180,E1 5613.498,E2 5613.498} C_VEL
LIN {X 0,Y 650.658,Z 859.31,A -85,B 0,C 180,E1 5618.951,E2 5618.951} C_VEL
LIN {X 0,Y 650.628,Z 859.31,A -85,B 0,C 180,E1 5624.31,E2 5624.31} C_VEL
LIN {X 0,Y 650.635,Z 859.31,A -85,B 0,C 180,E1 5629.299,E2 5629.299} C_VEL
LIN {X 0,Y 650.925,Z 859.318,A -85,B 0,C 180,E1 5635.002,E2 5635.002} C_VEL
LIN {X 0,Y 662.168,Z 884.977,A -85,B 0,C 180,E1 5635.853,E2 5635.853} C_VEL
LIN {X 0,Y 667.901,Z 896.404,A -85,B 0,C 180,E1 5636.248,E2 5636.248} C_VEL
LIN {X 0,Y 667.143,Z 945.956,A -85,B 0,C 180,E1 5636.999,E2 5636.999} C_VEL
LIN {X 0,Y 665.236,Z 990.18,A -85,B 0,C 180,E1 5638.209,E2 5638.209} C_VEL
LIN {X 0,Y 662.68,Z 1035.597,A -85,B 0,C 180,E1 5640.095,E2 5640.095} C_VEL
LIN {X 0,Y 659.863,Z 1077.71,A -85,B 0,C 180,E1 5642.508,E2 5642.508} C_VEL
LIN {X 0,Y 657.267,Z 1114.786,A -85,B 0,C 180,E1 5645.3,E2 5645.3} C_VEL
LIN {X 0,Y 655.186,Z 1145.858,A -85,B 0,C 180,E1 5648.282,E2 5648.282} C_VEL
LIN {X 0,Y 653.634,Z 1172.898,A -85,B 0,C 180,E1 5651.554,E2 5651.554} C_VEL
LIN {X 0,Y 652.465,Z 1196.127,A -85,B 0,C 180,E1 5655.199,E2 5655.199} C_VEL
LIN {X 0,Y 651.872,Z 1213.837,A -85,B 0,C 180,E1 5658.944,E2 5658.944} C_VEL
LIN {X 0,Y 651.552,Z 1226.068,A -85,B 0,C 180,E1 5662.651,E2 5662.651} C_VEL
LIN {X 0,Y 651.458,Z 1232.649,A -85,B 0,C 180,E1 5665.998,E2 5665.998} C_VEL
LIN {X 0,Y 651.473,Z 1235.5,A -85,B 0,C 180,E1 5670,E2 5670} C_VEL
LIN {X 0,Y 651.464,Z 1232.65,A -85,B 0,C 180,E1 5674.001,E2 5674.001} C_VEL
LIN {X 0,Y 651.509,Z 1226.069,A -85,B 0,C 180,E1 5677.349,E2 5677.349} C_VEL
LIN {X 0,Y 651.834,Z 1213.84,A -85,B 0,C 180,E1 5681.057,E2 5681.057} C_VEL
LIN {X 0,Y 652.456,Z 1196.126,A -85,B 0,C 180,E1 5684.801,E2 5684.801} C_VEL
LIN {X 0,Y 653.545,Z 1172.932,A -85,B 0,C 180,E1 5688.444,E2 5688.444} C_VEL
LIN {X 0,Y 655.35,Z 1142.592,A -85,B 0,C 180,E1 5692.075,E2 5692.075} C_VEL
LIN {X 0,Y 657.775,Z 1107.431,A -85,B 0,C 180,E1 5695.316,E2 5695.316} C_VEL
LIN {X 0,Y 660.378,Z 1069.764,A -85,B 0,C 180,E1 5698,E2 5698} C_VEL
LIN {X 0,Y 662.967,Z 1030.702,A -85,B 0,C 180,E1 5700.135,E2 5700.135} C_VEL
LIN {X 0,Y 665.403,Z 987.614,A -85,B 0,C 180,E1 5701.872,E2 5701.872} C_VEL
LIN {X 0,Y 667.243,Z 942.165,A -85,B 0,C 180,E1 5703.084,E2 5703.084} C_VEL
LIN {X 0,Y 667.31,Z 895.028,A -85,B 0,C 180,E1 5703.795,E2 5703.795} C_VEL
LIN {X 0,Y 651.074,Z 861.114,A -85,B 0,C 180,E1 5704.968,E2 5704.968} C_VEL
LIN {X 0,Y 650.876,Z 859.31,A -85,B 0,C 180,E1 5705.054,E2 5705.054} C_VEL
LIN {X 0,Y 650.733,Z 859.31,A -85,B 0,C 180,E1 5710.693,E2 5710.693} C_VEL
LIN {X 0,Y 650.782,Z 859.31,A -85,B 0,C 180,E1 5715.704,E2 5715.704} C_VEL
LIN {X 0,Y 650.645,Z 859.31,A -85,B 0,C 180,E1 5721.048,E2 5721.048} C_VEL
LIN {X 0,Y 650.709,Z 859.31,A -85,B 0,C 180,E1 5726.029,E2 5726.029} C_VEL
LIN {X 0,Y 650.847,Z 859.31,A -85,B 0,C 180,E1 5730.737,E2 5730.737} C_VEL
LIN {X 0,Y 650.948,Z 859.31,A -85,B 0,C 180,E1 5735.233,E2 5735.233} C_VEL
LIN {X 0,Y 650.975,Z 859.31,A -85,B 0,C 180,E1 5739.568,E2 5739.568} C_VEL
LIN {X 0,Y 651.012,Z 859.31,A -85,B 0,C 180,E1 5743.783,E2 5743.783} C_VEL
LIN {X 0,Y 651.084,Z 859.31,A -85,B 0,C 180,E1 5749.271,E2 5749.271} C_VEL
LIN {X 0,Y 651.228,Z 859.31,A -85,B 0,C 180,E1 5754.659,E2 5754.659} C_VEL
LIN {X 0,Y 651.31,Z 859.31,A -85,B 0,C 180,E1 5758.665,E2 5758.665} C_VEL
LIN {X 0,Y 651.295,Z 859.31,A -85,B 0,C 180,E1 5762.664,E2 5762.664} C_VEL
LIN {X 0,Y 651.144,Z 859.31,A -85,B 0,C 180,E1 5766.678,E2 5766.678} C_VEL
LIN {X 0,Y 651.091,Z 859.31,A -85,B 0,C 180,E1 5772.186,E2 5772.186} C_VEL
LIN {X 0,Y 651.041,Z 859.31,A -85,B 0,C 180,E1 5777.606,E2 5777.606} C_VEL
LIN {X 0,Y 650.916,Z 859.31,A -85,B 0,C 180,E1 5781.86,E2 5781.86} C_VEL
LIN {X 0,Y 650.896,Z 859.31,A -85,B 0,C 180,E1 5786.243,E2 5786.243} C_VEL
LIN {X 0,Y 650.794,Z 859.31,A -85,B 0,C 180,E1 5790.802,E2 5790.802} C_VEL
LIN {X 0,Y 650.763,Z 859.31,A -85,B 0,C 180,E1 5795.587,E2 5795.587} C_VEL
LIN {X 0,Y 650.668,Z 859.31,A -85,B 0,C 180,E1 5800.682,E2 5800.682} C_VEL
LIN {X 0,Y 650.622,Z 859.31,A -85,B 0,C 180,E1 5806.2,E2 5806.2} C_VEL
LIN {X 0,Y 650.697,Z 859.31,A -85,B 0,C 180,E1 5811.042,E2 5811.042} C_VEL
LIN {X 0,Y 650.835,Z 859.31,A -85,B 0,C 180,E1 5816.029,E2 5816.029} C_VEL
LIN {X 0,Y 650.823,Z 859.31,A -85,B 0,C 180,E1 5821.599,E2 5821.599} C_VEL
LIN {X 0,Y 663.571,Z 889.962,A -85,B 0,C 180,E1 5822.737,E2 5822.737} C_VEL
LIN {X 0,Y 662.573,Z 969.355,A -85,B 0,C 180,E1 5823.771,E2 5823.771} C_VEL
LIN {X 0,Y 661.06,Z 1008.505,A -85,B 0,C 180,E1 5824.805,E2 5824.805} C_VEL
LIN {X 0,Y 659.004,Z 1046.467,A -85,B 0,C 180,E1 5826.362,E2 5826.362} C_VEL
LIN {X 0,Y 656.829,Z 1082.141,A -85,B 0,C 180,E1 5828.437,E2 5828.437} C_VEL
LIN {X 0,Y 654.951,Z 1114.621,A -85,B 0,C 180,E1 5830.926,E2 5830.926} C_VEL
LIN {X 0,Y 653.491,Z 1142.034,A -85,B 0,C 180,E1 5833.671,E2 5833.671} C_VEL
LIN {X 0,Y 652.451,Z 1165.532,A -85,B 0,C 180,E1 5836.795,E2 5836.795} C_VEL
LIN {X 0,Y 651.854,Z 1182.997,A -85,B 0,C 180,E1 5839.96,E2 5839.96} C_VEL
LIN {X 0,Y 651.56,Z 1195.73,A -85,B 0,C 180,E1 5843.323,E2 5843.323} C_VEL
LIN {X 0,Y 651.525,Z 1202.013,A -85,B 0,C 180,E1 5845.999,E2 5845.999} C_VEL
LIN {X 0,Y 651.417,Z 1205.364,A -85,B 0,C 180,E1 5849.4,E2 5849.4} C_VEL
LIN {X 0,Y 651.516,Z 1203.84,A -85,B 0,C 180,E1 5852.666,E2 5852.666} C_VEL
LIN {X 0,Y 651.628,Z 1197.397,A -85,B 0,C 180,E1 5856.007,E2 5856.007} C_VEL
LIN {X 0,Y 651.797,Z 1185.654,A -85,B 0,C 180,E1 5859.366,E2 5859.366} C_VEL
LIN {X 0,Y 652.337,Z 1168.605,A -85,B 0,C 180,E1 5862.635,E2 5862.635} C_VEL
LIN {X 0,Y 653.306,Z 1145.599,A -85,B 0,C 180,E1 5865.822,E2 5865.822} C_VEL
LIN {X 0,Y 654.666,Z 1119.151,A -85,B 0,C 180,E1 5868.58,E2 5868.58} C_VEL
LIN {X 0,Y 656.41,Z 1087.586,A -85,B 0,C 180,E1 5871.093,E2 5871.093} C_VEL
LIN {X 0,Y 658.585,Z 1053.099,A -85,B 0,C 180,E1 5873.205,E2 5873.205} C_VEL
LIN {X 0,Y 660.603,Z 1017.551,A -85,B 0,C 180,E1 5874.783,E2 5874.783} C_VEL
LIN {X 0,Y 662.19,Z 980.518,A -85,B 0,C 180,E1 5875.898,E2 5875.898} C_VEL
LIN {X 0,Y 663.024,Z 940.448,A -85,B 0,C 180,E1 5876.58,E2 5876.58} C_VEL
LIN {X 0,Y 662.828,Z 888.096,A -85,B 0,C 180,E1 5877.227,E2 5877.227} C_VEL
LIN {X 0,Y 650.856,Z 859.31,A -85,B 0,C 180,E1 5878.333,E2 5878.333} C_VEL
LIN {X 0,Y 650.834,Z 859.31,A -85,B 0,C 180,E1 5883.971,E2 5883.971} C_VEL
LIN {X 0,Y 650.712,Z 859.31,A -85,B 0,C 180,E1 5888.958,E2 5888.958} C_VEL
LIN {X 0,Y 650.608,Z 859.31,A -85,B 0,C 180,E1 5894.324,E2 5894.324} C_VEL
LIN {X 0,Y 650.658,Z 859.31,A -85,B 0,C 180,E1 5899.317,E2 5899.317} C_VEL
LIN {X 0,Y 650.839,Z 859.31,A -85,B 0,C 180,E1 5904.575,E2 5904.575} C_VEL
LIN {X 0,Y 650.792,Z 859.31,A -85,B 0,C 180,E1 5909.486,E2 5909.486} C_VEL
LIN {X 0,Y 650.921,Z 859.31,A -85,B 0,C 180,E1 5913.759,E2 5913.759} C_VEL
LIN {X 0,Y 650.97,Z 859.31,A -85,B 0,C 180,E1 5918.607,E2 5918.607} C_VEL
LIN {X 0,Y 650.774,Z 859.31,A -85,B 0,C 180,E1 5923.781,E2 5923.781} C_VEL
LIN {X 0,Y 651.121,Z 859.31,A -85,B 0,C 180,E1 5929.275,E2 5929.275} C_VEL
LIN {X 0,Y 651.241,Z 859.31,A -85,B 0,C 180,E1 5934.663,E2 5934.663} C_VEL
LIN {X 0,Y 651.365,Z 859.31,A -85,B 0,C 180,E1 5940.002,E2 5940.002} C_VEL
LIN {X 0,Y 651.378,Z 859.31,A -85,B 0,C 180,E1 5945.34,E2 5945.34} C_VEL
LIN {X 0,Y 651.04,Z 859.31,A -85,B 0,C 180,E1 5950.73,E2 5950.73} C_VEL
LIN {X 0,Y 651.048,Z 859.31,A -85,B 0,C 180,E1 5956.216,E2 5956.216} C_VEL
LIN {X 0,Y 650.994,Z 859.31,A -85,B 0,C 180,E1 5961.398,E2 5961.398} C_VEL
LIN {X 0,Y 650.925,Z 859.31,A -85,B 0,C 180,E1 5966.245,E2 5966.245} C_VEL
LIN {X 0,Y 650.803,Z 859.31,A -85,B 0,C 180,E1 5970.806,E2 5970.806} C_VEL
LIN {X 0,Y 650.712,Z 859.31,A -85,B 0,C 180,E1 5973.498,E2 5973.498} C_VEL
LIN {X 0,Y 648.209,Z 859.31,A -85,B 0,C 180,E1 5974.627,E2 5974.627} C_VEL
LIN {X 0,Y 642.862,Z 859.31,A -85,B 0,C 180,E1 5976.313,E2 5976.313} C_VEL
LIN {X 0,Y 642.767,Z 859.31,A -85,B 0,C 180,E1 5976.508,E2 5976.508} C_VEL
LIN {X 0,Y 642.729,Z 859.31,A -85,B 0,C 180,E1 5981.299,E2 5981.299} C_VEL
LIN {X 0,Y 642.709,Z 859.31,A -85,B 0,C 180,E1 5986.946,E2 5986.946} C_VEL
LIN {X 0,Y 642.807,Z 859.31,A -85,B 0,C 180,E1 5992.2,E2 5992.2} C_VEL
LIN {X 0,Y 642.983,Z 859.31,A -85,B 0,C 180,E1 5994.609,E2 5994.609} C_VEL
LIN {X 0,Y 656.169,Z 889.415,A -85,B 0,C 180,E1 5995.628,E2 5995.628} C_VEL
LIN {X 0,Y 660.931,Z 899.437,A -85,B 0,C 180,E1 5995.969,E2 5995.969} C_VEL
LIN {X 0,Y 660.062,Z 946.719,A -85,B 0,C 180,E1 5996.707,E2 5996.707} C_VEL
LIN {X 0,Y 658.259,Z 991.088,A -85,B 0,C 180,E1 5997.9,E2 5997.9} C_VEL
LIN {X 0,Y 656.104,Z 1029.628,A -85,B 0,C 180,E1 5999.463,E2 5999.463} C_VEL
LIN {X 0,Y 653.429,Z 1068.339,A -85,B 0,C 180,E1 6001.58,E2 6001.58} C_VEL
LIN {X 0,Y 650.565,Z 1106.371,A -85,B 0,C 180,E1 6004.29,E2 6004.29} C_VEL
LIN {X 0,Y 647.874,Z 1141.837,A -85,B 0,C 180,E1 6007.572,E2 6007.572} C_VEL
LIN {X 0,Y 645.951,Z 1172.496,A -85,B 0,C 180,E1 6011.268,E2 6011.268} C_VEL
LIN {X 0,Y 644.662,Z 1196.126,A -85,B 0,C 180,E1 6015.015,E2 6015.015} C_VEL
LIN {X 0,Y 644.023,Z 1213.836,A -85,B 0,C 180,E1 6018.807,E2 6018.807} C_VEL
LIN {X 0,Y 643.678,Z 1226.068,A -85,B 0,C 180,E1 6022.56,E2 6022.56} C_VEL
LIN {X 0,Y 643.56,Z 1232.649,A -85,B 0,C 180,E1 6025.949,E2 6025.949} C_VEL
LIN {X 0,Y 643.6,Z 1235.5,A -85,B 0,C 180,E1 6030,E2 6030} C_VEL
LIN {X 0,Y 643.565,Z 1232.65,A -85,B 0,C 180,E1 6034.05,E2 6034.05} C_VEL
LIN {X 0,Y 643.633,Z 1226.068,A -85,B 0,C 180,E1 6037.44,E2 6037.44} C_VEL
LIN {X 0,Y 643.99,Z 1213.839,A -85,B 0,C 180,E1 6041.193,E2 6041.193} C_VEL
LIN {X 0,Y 644.649,Z 1196.124,A -85,B 0,C 180,E1 6044.985,E2 6044.985} C_VEL
LIN {X 0,Y 645.905,Z 1172.498,A -85,B 0,C 180,E1 6048.733,E2 6048.733} C_VEL
LIN {X 0,Y 647.851,Z 1141.878,A -85,B 0,C 180,E1 6052.425,E2 6052.425} C_VEL
LIN {X 0,Y 650.552,Z 1106.378,A -85,B 0,C 180,E1 6055.71,E2 6055.71} C_VEL
LIN {X 0,Y 653.558,Z 1066.272,A -85,B 0,C 180,E1 6058.555,E2 6058.555} C_VEL
LIN {X 0,Y 656.453,Z 1024.301,A -85,B 0,C 180,E1 6060.788,E2 6060.788} C_VEL
LIN {X 0,Y 658.528,Z 986.041,A -85,B 0,C 180,E1 6062.259,E2 6062.259} C_VEL
LIN {X 0,Y 660.228,Z 940.692,A -85,B 0,C 180,E1 6063.423,E2 6063.423} C_VEL
LIN {X 0,Y 660.299,Z 897.529,A -85,B 0,C 180,E1 6064.082,E2 6064.082} C_VEL
LIN {X 0,Y 643.177,Z 861.143,A -85,B 0,C 180,E1 6065.362,E2 6065.362} C_VEL
LIN {X 0,Y 642.928,Z 859.31,A -85,B 0,C 180,E1 6065.437,E2 6065.437} C_VEL
LIN {X 0,Y 642.829,Z 859.31,A -85,B 0,C 180,E1 6071.301,E2 6071.301} C_VEL
LIN {X 0,Y 642.806,Z 859.31,A -85,B 0,C 180,E1 6076.95,E2 6076.95} C_VEL
LIN {X 0,Y 642.718,Z 859.31,A -85,B 0,C 180,E1 6082.204,E2 6082.204} C_VEL
LIN {X 0,Y 642.817,Z 859.31,A -85,B 0,C 180,E1 6087.176,E2 6087.176} C_VEL
LIN {X 0,Y 642.959,Z 859.31,A -85,B 0,C 180,E1 6091.884,E2 6091.884} C_VEL
LIN {X 0,Y 643.073,Z 859.31,A -85,B 0,C 180,E1 6096.775,E2 6096.775} C_VEL
LIN {X 0,Y 643.104,Z 859.31,A -85,B 0,C 180,E1 6102.166,E2 6102.166} C_VEL
LIN {X 0,Y 643.1,Z 859.31,A -85,B 0,C 180,E1 6107.758,E2 6107.758} C_VEL
LIN {X 0,Y 643.347,Z 859.31,A -85,B 0,C 180,E1 6113.237,E2 6113.237} C_VEL
LIN {X 0,Y 643.41,Z 859.31,A -85,B 0,C 180,E1 6118.649,E2 6118.649} C_VEL
LIN {X 0,Y 643.393,Z 859.31,A -85,B 0,C 180,E1 6122.697,E2 6122.697} C_VEL
LIN {X 0,Y 643.235,Z 859.31,A -85,B 0,C 180,E1 6126.761,E2 6126.761} C_VEL
LIN {X 0,Y 643.206,Z 859.31,A -85,B 0,C 180,E1 6132.236,E2 6132.236} C_VEL
LIN {X 0,Y 643.113,Z 859.31,A -85,B 0,C 180,E1 6137.83,E2 6137.83} C_VEL
LIN {X 0,Y 643.007,Z 859.31,A -85,B 0,C 180,E1 6143.211,E2 6143.211} C_VEL
LIN {X 0,Y 642.913,Z 859.31,A -85,B 0,C 180,E1 6148.114,E2 6148.114} C_VEL
LIN {X 0,Y 642.845,Z 859.31,A -85,B 0,C 180,E1 6152.818,E2 6152.818} C_VEL
LIN {X 0,Y 642.772,Z 859.31,A -85,B 0,C 180,E1 6157.788,E2 6157.788} C_VEL
LIN {X 0,Y 642.704,Z 859.31,A -85,B 0,C 180,E1 6163.119,E2 6163.119} C_VEL
LIN {X 0,Y 642.749,Z 859.31,A -85,B 0,C 180,E1 6168.953,E2 6168.953} C_VEL
LIN {X 0,Y 642.85,Z 859.31,A -85,B 0,C 180,E1 6173.894,E2 6173.894} C_VEL
LIN {X 0,Y 642.795,Z 859.31,A -85,B 0,C 180,E1 6178.761,E2 6178.761} C_VEL
LIN {X 0,Y 642.899,Z 859.351,A -85,B 0,C 180,E1 6181.151,E2 6181.151} C_VEL
LIN {X 0,Y 656.772,Z 891.447,A -85,B 0,C 180,E1 6182.369,E2 6182.369} C_VEL
LIN {X 0,Y 655.93,Z 969.6,A -85,B 0,C 180,E1 6183.4,E2 6183.4} C_VEL
LIN {X 0,Y 654.287,Z 1008.713,A -85,B 0,C 180,E1 6184.439,E2 6184.439} C_VEL
LIN {X 0,Y 652.065,Z 1046.403,A -85,B 0,C 180,E1 6186.004,E2 6186.004} C_VEL
LIN {X 0,Y 649.62,Z 1082.999,A -85,B 0,C 180,E1 6188.164,E2 6188.164} C_VEL
LIN {X 0,Y 647.39,Z 1114.83,A -85,B 0,C 180,E1 6190.694,E2 6190.694} C_VEL
LIN {X 0,Y 645.678,Z 1143.489,A -85,B 0,C 180,E1 6193.643,E2 6193.643} C_VEL
LIN {X 0,Y 644.604,Z 1166.243,A -85,B 0,C 180,E1 6196.745,E2 6196.745} C_VEL
LIN {X 0,Y 644.015,Z 1182.994,A -85,B 0,C 180,E1 6199.836,E2 6199.836} C_VEL
LIN {X 0,Y 643.677,Z 1195.728,A -85,B 0,C 180,E1 6203.24,E2 6203.24} C_VEL
LIN {X 0,Y 643.629,Z 1202.011,A -85,B 0,C 180,E1 6205.95,E2 6205.95} C_VEL
LIN {X 0,Y 643.563,Z 1205.119,A -85,B 0,C 180,E1 6208.651,E2 6208.651} C_VEL
LIN {X 0,Y 643.62,Z 1205.049,A -85,B 0,C 180,E1 6211.349,E2 6211.349} C_VEL
LIN {X 0,Y 643.727,Z 1200.625,A -85,B 0,C 180,E1 6214.726,E2 6214.726} C_VEL
LIN {X 0,Y 643.837,Z 1191.039,A -85,B 0,C 180,E1 6218.118,E2 6218.118} C_VEL
LIN {X 0,Y 644.331,Z 1175.817,A -85,B 0,C 180,E1 6221.531,E2 6221.531} C_VEL
LIN {X 0,Y 645.069,Z 1155.149,A -85,B 0,C 180,E1 6224.801,E2 6224.801} C_VEL
LIN {X 0,Y 646.391,Z 1130.141,A -85,B 0,C 180,E1 6227.743,E2 6227.743} C_VEL
LIN {X 0,Y 648.47,Z 1098.21,A -85,B 0,C 180,E1 6230.626,E2 6230.626} C_VEL
LIN {X 0,Y 650.794,Z 1064.602,A -85,B 0,C 180,E1 6232.916,E2 6232.916} C_VEL
LIN {X 0,Y 653.1,Z 1029.332,A -85,B 0,C 180,E1 6234.685,E2 6234.685} C_VEL
LIN {X 0,Y 655.026,Z 992.96,A -85,B 0,C 180,E1 6235.953,E2 6235.953} C_VEL
LIN {X 0,Y 656.257,Z 954.842,A -85,B 0,C 180,E1 6236.765,E2 6236.765} C_VEL
LIN {X 0,Y 656.192,Z 890.062,A -85,B 0,C 180,E1 6237.59,E2 6237.59} C_VEL
LIN {X 0,Y 642.913,Z 859.31,A -85,B 0,C 180,E1 6238.814,E2 6238.814} C_VEL
LIN {X 0,Y 642.893,Z 859.31,A -85,B 0,C 180,E1 6244.45,E2 6244.45} C_VEL
LIN {X 0,Y 642.802,Z 859.31,A -85,B 0,C 180,E1 6249.53,E2 6249.53} C_VEL
LIN {X 0,Y 642.683,Z 859.31,A -85,B 0,C 180,E1 6255.018,E2 6255.018} C_VEL
LIN {X 0,Y 642.749,Z 859.31,A -85,B 0,C 180,E1 6260.481,E2 6260.481} C_VEL
LIN {X 0,Y 642.898,Z 859.31,A -85,B 0,C 180,E1 6265.583,E2 6265.583} C_VEL
LIN {X 0,Y 642.916,Z 859.31,A -85,B 0,C 180,E1 6270.699,E2 6270.699} C_VEL
LIN {X 0,Y 643.007,Z 859.31,A -85,B 0,C 180,E1 6274.91,E2 6274.91} C_VEL
LIN {X 0,Y 643.01,Z 859.31,A -85,B 0,C 180,E1 6279.307,E2 6279.307} C_VEL
LIN {X 0,Y 642.971,Z 859.31,A -85,B 0,C 180,E1 6285.072,E2 6285.072} C_VEL
LIN {X 0,Y 643.257,Z 859.31,A -85,B 0,C 180,E1 6290.513,E2 6290.513} C_VEL
LIN {X 0,Y 643.407,Z 859.31,A -85,B 0,C 180,E1 6295.951,E2 6295.951} C_VEL
LIN {X 0,Y 643.58,Z 859.31,A -85,B 0,C 180,E1 6301.351,E2 6301.351} C_VEL
LIN {X 0,Y 643.238,Z 859.31,A -85,B 0,C 180,E1 6306.764,E2 6306.764} C_VEL
LIN {X 0,Y 643.156,Z 859.31,A -85,B 0,C 180,E1 6312.241,E2 6312.241} C_VEL
LIN {X 0,Y 643.139,Z 859.31,A -85,B 0,C 180,E1 6317.833,E2 6317.833} C_VEL
LIN {X 0,Y 643.026,Z 859.31,A -85,B 0,C 180,E1 6323.214,E2 6323.214} C_VEL
LIN {X 0,Y 642.944,Z 859.31,A -85,B 0,C 180,E1 6328.117,E2 6328.117} C_VEL
LIN {X 0,Y 642.765,Z 859.31,A -85,B 0,C 180,E1 6333.496,E2 6333.496} C_VEL
LIN {X 0,Y 642.767,Z 859.31,A -85,B 0,C 180,E1 6336.508,E2 6336.508} C_VEL
LIN {X 0,Y 641.489,Z 859.31,A -85,B 0,C 180,E1 6337.28,E2 6337.28} C_VEL
LIN {X 0,Y 634.835,Z 859.31,A -85,B 0,C 180,E1 6339.378,E2 6339.378} C_VEL
LIN {X 0,Y 634.747,Z 859.31,A -85,B 0,C 180,E1 6339.576,E2 6339.576} C_VEL
LIN {X 0,Y 634.723,Z 859.31,A -85,B 0,C 180,E1 6344.258,E2 6344.258} C_VEL
LIN {X 0,Y 634.79,Z 859.31,A -85,B 0,C 180,E1 6349.871,E2 6349.871} C_VEL
LIN {X 0,Y 635.025,Z 859.31,A -85,B 0,C 180,E1 6354.206,E2 6354.206} C_VEL
LIN {X 0,Y 650.027,Z 893.502,A -85,B 0,C 180,E1 6355.386,E2 6355.386} C_VEL
LIN {X 0,Y 653.942,Z 902.568,A -85,B 0,C 180,E1 6355.684,E2 6355.684} C_VEL
LIN {X 0,Y 652.946,Z 948.877,A -85,B 0,C 180,E1 6356.44,E2 6356.44} C_VEL
LIN {X 0,Y 651.029,Z 992.117,A -85,B 0,C 180,E1 6357.633,E2 6357.633} C_VEL
LIN {X 0,Y 648.637,Z 1036.814,A -85,B 0,C 180,E1 6359.465,E2 6359.465} C_VEL
LIN {X 0,Y 645.789,Z 1074.689,A -85,B 0,C 180,E1 6361.649,E2 6361.649} C_VEL
LIN {X 0,Y 642.821,Z 1110.576,A -85,B 0,C 180,E1 6364.332,E2 6364.332} C_VEL
LIN {X 0,Y 640.223,Z 1143.253,A -85,B 0,C 180,E1 6367.45,E2 6367.45} C_VEL
LIN {X 0,Y 638.232,Z 1172.961,A -85,B 0,C 180,E1 6371.101,E2 6371.101} C_VEL
LIN {X 0,Y 636.884,Z 1196.125,A -85,B 0,C 180,E1 6374.828,E2 6374.828} C_VEL
LIN {X 0,Y 636.15,Z 1213.836,A -85,B 0,C 180,E1 6378.667,E2 6378.667} C_VEL
LIN {X 0,Y 635.787,Z 1226.068,A -85,B 0,C 180,E1 6382.468,E2 6382.468} C_VEL
LIN {X 0,Y 635.682,Z 1232.648,A -85,B 0,C 180,E1 6385.899,E2 6385.899} C_VEL
LIN {X 0,Y 635.702,Z 1235.5,A -85,B 0,C 180,E1 6390,E2 6390} C_VEL
LIN {X 0,Y 635.687,Z 1232.649,A -85,B 0,C 180,E1 6394.101,E2 6394.101} C_VEL
LIN {X 0,Y 635.74,Z 1226.068,A -85,B 0,C 180,E1 6397.533,E2 6397.533} C_VEL
LIN {X 0,Y 636.121,Z 1213.839,A -85,B 0,C 180,E1 6401.333,E2 6401.333} C_VEL
LIN {X 0,Y 636.861,Z 1196.123,A -85,B 0,C 180,E1 6405.172,E2 6405.172} C_VEL
LIN {X 0,Y 638.301,Z 1171.743,A -85,B 0,C 180,E1 6409.068,E2 6409.068} C_VEL
LIN {X 0,Y 640.305,Z 1142.16,A -85,B 0,C 180,E1 6412.672,E2 6412.672} C_VEL
LIN {X 0,Y 643.235,Z 1106.376,A -85,B 0,C 180,E1 6416.024,E2 6416.024} C_VEL
LIN {X 0,Y 646.421,Z 1066.795,A -85,B 0,C 180,E1 6418.864,E2 6418.864} C_VEL
LIN {X 0,Y 648.904,Z 1031.449,A -85,B 0,C 180,E1 6420.784,E2 6420.784} C_VEL
LIN {X 0,Y 651.294,Z 988.62,A -85,B 0,C 180,E1 6422.482,E2 6422.482} C_VEL
LIN {X 0,Y 653.188,Z 940.997,A -85,B 0,C 180,E1 6423.734,E2 6423.734} C_VEL
LIN {X 0,Y 653.328,Z 900.094,A -85,B 0,C 180,E1 6424.375,E2 6424.375} C_VEL
LIN {X 0,Y 635.334,Z 861.497,A -85,B 0,C 180,E1 6425.75,E2 6425.75} C_VEL
LIN {X 0,Y 634.989,Z 859.31,A -85,B 0,C 180,E1 6425.853,E2 6425.853} C_VEL
LIN {X 0,Y 634.847,Z 859.31,A -85,B 0,C 180,E1 6430.215,E2 6430.215} C_VEL
LIN {X 0,Y 634.888,Z 859.31,A -85,B 0,C 180,E1 6435.726,E2 6435.726} C_VEL
LIN {X 0,Y 634.828,Z 859.31,A -85,B 0,C 180,E1 6441.65,E2 6441.65} C_VEL
LIN {X 0,Y 634.853,Z 859.31,A -85,B 0,C 180,E1 6446.711,E2 6446.711} C_VEL
LIN {X 0,Y 635.067,Z 859.31,A -85,B 0,C 180,E1 6451.986,E2 6451.986} C_VEL
LIN {X 0,Y 635.122,Z 859.31,A -85,B 0,C 180,E1 6457.563,E2 6457.563} C_VEL
LIN {X 0,Y 635.172,Z 859.31,A -85,B 0,C 180,E1 6462.602,E2 6462.602} C_VEL
LIN {X 0,Y 635.212,Z 859.31,A -85,B 0,C 180,E1 6467.973,E2 6467.973} C_VEL
LIN {X 0,Y 635.444,Z 859.31,A -85,B 0,C 180,E1 6473.152,E2 6473.152} C_VEL
LIN {X 0,Y 635.509,Z 859.31,A -85,B 0,C 180,E1 6478.632,E2 6478.632} C_VEL
LIN {X 0,Y 635.501,Z 859.31,A -85,B 0,C 180,E1 6482.731,E2 6482.731} C_VEL
LIN {X 0,Y 635.326,Z 859.31,A -85,B 0,C 180,E1 6486.845,E2 6486.845} C_VEL
LIN {X 0,Y 635.285,Z 859.31,A -85,B 0,C 180,E1 6492.391,E2 6492.391} C_VEL
LIN {X 0,Y 635.19,Z 859.31,A -85,B 0,C 180,E1 6498.06,E2 6498.06} C_VEL
LIN {X 0,Y 635.067,Z 859.31,A -85,B 0,C 180,E1 6502.435,E2 6502.435} C_VEL
LIN {X 0,Y 635.028,Z 859.31,A -85,B 0,C 180,E1 6508.008,E2 6508.008} C_VEL
LIN {X 0,Y 634.885,Z 859.31,A -85,B 0,C 180,E1 6513.348,E2 6513.348} C_VEL
LIN {X 0,Y 634.862,Z 859.31,A -85,B 0,C 180,E1 6518.343,E2 6518.343} C_VEL
LIN {X 0,Y 634.718,Z 859.31,A -85,B 0,C 180,E1 6523.798,E2 6523.798} C_VEL
LIN {X 0,Y 634.816,Z 859.31,A -85,B 0,C 180,E1 6529.782,E2 6529.782} C_VEL
LIN {X 0,Y 634.923,Z 859.31,A -85,B 0,C 180,E1 6535.056,E2 6535.056} C_VEL
LIN {X 0,Y 634.975,Z 859.31,A -85,B 0,C 180,E1 6540.662,E2 6540.662} C_VEL
LIN {X 0,Y 650.311,Z 893.809,A -85,B 0,C 180,E1 6542.013,E2 6542.013} C_VEL
LIN {X 0,Y 649.323,Z 969.675,A -85,B 0,C 180,E1 6543.016,E2 6543.016} C_VEL
LIN {X 0,Y 647.596,Z 1008.41,A -85,B 0,C 180,E1 6544.051,E2 6544.051} C_VEL
LIN {X 0,Y 645.184,Z 1046.492,A -85,B 0,C 180,E1 6545.64,E2 6545.64} C_VEL
LIN {X 0,Y 642.565,Z 1082.078,A -85,B 0,C 180,E1 6547.751,E2 6547.751} C_VEL
LIN {X 0,Y 640.071,Z 1113.862,A -85,B 0,C 180,E1 6550.285,E2 6550.285} C_VEL
LIN {X 0,Y 638.139,Z 1142.163,A -85,B 0,C 180,E1 6553.267,E2 6553.267} C_VEL
LIN {X 0,Y 636.812,Z 1166.194,A -85,B 0,C 180,E1 6556.573,E2 6556.573} C_VEL
LIN {X 0,Y 636.18,Z 1182.992,A -85,B 0,C 180,E1 6559.71,E2 6559.71} C_VEL
LIN {X 0,Y 635.799,Z 1195.726,A -85,B 0,C 180,E1 6563.156,E2 6563.156} C_VEL
LIN {X 0,Y 635.742,Z 1202.01,A -85,B 0,C 180,E1 6565.9,E2 6565.9} C_VEL
LIN {X 0,Y 635.662,Z 1205.119,A -85,B 0,C 180,E1 6568.634,E2 6568.634} C_VEL
LIN {X 0,Y 635.73,Z 1205.05,A -85,B 0,C 180,E1 6571.366,E2 6571.366} C_VEL
LIN {X 0,Y 635.831,Z 1200.626,A -85,B 0,C 180,E1 6574.785,E2 6574.785} C_VEL
LIN {X 0,Y 635.98,Z 1191.041,A -85,B 0,C 180,E1 6578.219,E2 6578.219} C_VEL
LIN {X 0,Y 636.484,Z 1175.821,A -85,B 0,C 180,E1 6581.675,E2 6581.675} C_VEL
LIN {X 0,Y 637.314,Z 1155.152,A -85,B 0,C 180,E1 6584.985,E2 6584.985} C_VEL
LIN {X 0,Y 639.032,Z 1127.53,A -85,B 0,C 180,E1 6588.289,E2 6588.289} C_VEL
LIN {X 0,Y 641.229,Z 1097.997,A -85,B 0,C 180,E1 6590.974,E2 6590.974} C_VEL
LIN {X 0,Y 643.745,Z 1065.495,A -85,B 0,C 180,E1 6593.223,E2 6593.223} C_VEL
LIN {X 0,Y 646.249,Z 1030.09,A -85,B 0,C 180,E1 6595.028,E2 6595.028} C_VEL
LIN {X 0,Y 648.345,Z 993.482,A -85,B 0,C 180,E1 6596.32,E2 6596.32} C_VEL
LIN {X 0,Y 649.657,Z 955.169,A -85,B 0,C 180,E1 6597.146,E2 6597.146} C_VEL
LIN {X 0,Y 649.523,Z 892.097,A -85,B 0,C 180,E1 6597.948,E2 6597.948} C_VEL
LIN {X 0,Y 635.003,Z 859.31,A -85,B 0,C 180,E1 6599.282,E2 6599.282} C_VEL
LIN {X 0,Y 634.92,Z 859.31,A -85,B 0,C 180,E1 6604.945,E2 6604.945} C_VEL
LIN {X 0,Y 634.828,Z 859.31,A -85,B 0,C 180,E1 6610.219,E2 6610.219} C_VEL
LIN {X 0,Y 634.715,Z 859.31,A -85,B 0,C 180,E1 6616.202,E2 6616.202} C_VEL
LIN {X 0,Y 634.887,Z 859.31,A -85,B 0,C 180,E1 6621.964,E2 6621.964} C_VEL
LIN {X 0,Y 634.906,Z 859.31,A -85,B 0,C 180,E1 6626.719,E2 6626.719} C_VEL
LIN {X 0,Y 635.03,Z 859.31,A -85,B 0,C 180,E1 6631.993,E2 6631.993} C_VEL
LIN {X 0,Y 635.095,Z 859.31,A -85,B 0,C 180,E1 6637.566,E2 6637.566} C_VEL
LIN {X 0,Y 634.935,Z 859.31,A -85,B 0,C 180,E1 6643.365,E2 6643.365} C_VEL
LIN {X 0,Y 635.294,Z 859.31,A -85,B 0,C 180,E1 6649.005,E2 6649.005} C_VEL
LIN {X 0,Y 635.431,Z 859.31,A -85,B 0,C 180,E1 6654.53,E2 6654.53} C_VEL
LIN {X 0,Y 635.513,Z 859.31,A -85,B 0,C 180,E1 6658.636,E2 6658.636} C_VEL
LIN {X 0,Y 635.502,Z 859.31,A -85,B 0,C 180,E1 6662.735,E2 6662.735} C_VEL
LIN {X 0,Y 635.328,Z 859.31,A -85,B 0,C 180,E1 6666.849,E2 6666.849} C_VEL
LIN {X 0,Y 635.254,Z 859.31,A -85,B 0,C 180,E1 6672.395,E2 6672.395} C_VEL
LIN {X 0,Y 635.216,Z 859.31,A -85,B 0,C 180,E1 6678.063,E2 6678.063} C_VEL
LIN {X 0,Y 635.11,Z 859.31,A -85,B 0,C 180,E1 6682.437,E2 6682.437} C_VEL
LIN {X 0,Y 635.051,Z 859.31,A -85,B 0,C 180,E1 6688.011,E2 6688.011} C_VEL
LIN {X 0,Y 634.872,Z 859.31,A -85,B 0,C 180,E1 6693.345,E2 6693.345} C_VEL
LIN {X 0,Y 634.856,Z 859.31,A -85,B 0,C 180,E1 6698.348,E2 6698.348} C_VEL
LIN {X 0,Y 634.747,Z 859.31,A -85,B 0,C 180,E1 6699.576,E2 6699.576} C_VEL
LIN {X 0,Y 633.515,Z 859.31,A -85,B 0,C 180,E1 6700.359,E2 6700.359} C_VEL
LIN {X 0,Y 626.91,Z 859.31,A -85,B 0,C 180,E1 6702.484,E2 6702.484} C_VEL
LIN {X 0,Y 626.808,Z 859.31,A -85,B 0,C 180,E1 6702.685,E2 6702.685} C_VEL
LIN {X 0,Y 626.808,Z 859.31,A -85,B 0,C 180,E1 6707.398,E2 6707.398} C_VEL
LIN {X 0,Y 626.994,Z 859.31,A -85,B 0,C 180,E1 6712.878,E2 6712.878} C_VEL
LIN {X 0,Y 627.075,Z 859.31,A -85,B 0,C 180,E1 6713.789,E2 6713.789} C_VEL
LIN {X 0,Y 643.967,Z 897.812,A -85,B 0,C 180,E1 6715.152,E2 6715.152} C_VEL
LIN {X 0,Y 646.976,Z 904.422,A -85,B 0,C 180,E1 6715.377,E2 6715.377} C_VEL
LIN {X 0,Y 645.753,Z 952.23,A -85,B 0,C 180,E1 6716.192,E2 6716.192} C_VEL
LIN {X 0,Y 643.645,Z 996.007,A -85,B 0,C 180,E1 6717.463,E2 6717.463} C_VEL
LIN {X 0,Y 641.303,Z 1037.672,A -85,B 0,C 180,E1 6719.22,E2 6719.22} C_VEL
LIN {X 0,Y 638.335,Z 1078.356,A -85,B 0,C 180,E1 6721.544,E2 6721.544} C_VEL
LIN {X 0,Y 634.988,Z 1116.883,A -85,B 0,C 180,E1 6724.561,E2 6724.561} C_VEL
LIN {X 0,Y 632.299,Z 1149.055,A -85,B 0,C 180,E1 6727.824,E2 6727.824} C_VEL
LIN {X 0,Y 630.323,Z 1176.114,A -85,B 0,C 180,E1 6731.329,E2 6731.329} C_VEL
LIN {X 0,Y 628.967,Z 1198.043,A -85,B 0,C 180,E1 6734.99,E2 6734.99} C_VEL
LIN {X 0,Y 628.159,Z 1216.511,A -85,B 0,C 180,E1 6739.225,E2 6739.225} C_VEL
LIN {X 0,Y 627.823,Z 1227.635,A -85,B 0,C 180,E1 6743.069,E2 6743.069} C_VEL
LIN {X 0,Y 627.785,Z 1232.648,A -85,B 0,C 180,E1 6745.847,E2 6745.847} C_VEL
LIN {X 0,Y 627.802,Z 1235.5,A -85,B 0,C 180,E1 6750,E2 6750} C_VEL
LIN {X 0,Y 627.789,Z 1232.649,A -85,B 0,C 180,E1 6754.152,E2 6754.152} C_VEL
LIN {X 0,Y 627.857,Z 1226.068,A -85,B 0,C 180,E1 6757.628,E2 6757.628} C_VEL
LIN {X 0,Y 628.259,Z 1213.838,A -85,B 0,C 180,E1 6761.477,E2 6761.477} C_VEL
LIN {X 0,Y 629.08,Z 1196.121,A -85,B 0,C 180,E1 6765.365,E2 6765.365} C_VEL
LIN {X 0,Y 630.632,Z 1171.861,A -85,B 0,C 180,E1 6769.292,E2 6769.292} C_VEL
LIN {X 0,Y 632.843,Z 1142.161,A -85,B 0,C 180,E1 6772.954,E2 6772.954} C_VEL
LIN {X 0,Y 635.836,Z 1107.373,A -85,B 0,C 180,E1 6776.26,E2 6776.26} C_VEL
LIN {X 0,Y 638.843,Z 1071.841,A -85,B 0,C 180,E1 6778.873,E2 6778.873} C_VEL
LIN {X 0,Y 641.601,Z 1032.23,A -85,B 0,C 180,E1 6781.041,E2 6781.041} C_VEL
LIN {X 0,Y 644.177,Z 988.105,A -85,B 0,C 180,E1 6782.809,E2 6782.809} C_VEL
LIN {X 0,Y 646.177,Z 940.636,A -85,B 0,C 180,E1 6784.063,E2 6784.063} C_VEL
LIN {X 0,Y 646.45,Z 902.57,A -85,B 0,C 180,E1 6784.673,E2 6784.673} C_VEL
LIN {X 0,Y 628.934,Z 864.964,A -85,B 0,C 180,E1 6786.028,E2 6786.028} C_VEL
LIN {X 0,Y 627.051,Z 859.31,A -85,B 0,C 180,E1 6786.211,E2 6786.211} C_VEL
LIN {X 0,Y 626.918,Z 859.31,A -85,B 0,C 180,E1 6791.486,E2 6791.486} C_VEL
LIN {X 0,Y 626.932,Z 859.31,A -85,B 0,C 180,E1 6796.477,E2 6796.477} C_VEL
LIN {X 0,Y 626.858,Z 859.31,A -85,B 0,C 180,E1 6801.071,E2 6801.071} C_VEL
LIN {X 0,Y 626.908,Z 859.31,A -85,B 0,C 180,E1 6806.233,E2 6806.233} C_VEL
LIN {X 0,Y 627.085,Z 859.31,A -85,B 0,C 180,E1 6811.106,E2 6811.106} C_VEL
LIN {X 0,Y 627.158,Z 859.31,A -85,B 0,C 180,E1 6816.653,E2 6816.653} C_VEL
LIN {X 0,Y 627.254,Z 859.31,A -85,B 0,C 180,E1 6821.7,E2 6821.7} C_VEL
LIN {X 0,Y 627.248,Z 859.31,A -85,B 0,C 180,E1 6827.444,E2 6827.444} C_VEL
LIN {X 0,Y 627.527,Z 859.31,A -85,B 0,C 180,E1 6833.065,E2 6833.065} C_VEL
LIN {X 0,Y 627.609,Z 859.31,A -85,B 0,C 180,E1 6838.615,E2 6838.615} C_VEL
LIN {X 0,Y 627.598,Z 859.31,A -85,B 0,C 180,E1 6842.765,E2 6842.765} C_VEL
LIN {X 0,Y 627.439,Z 859.31,A -85,B 0,C 180,E1 6848.042,E2 6848.042} C_VEL
LIN {X 0,Y 627.361,Z 859.31,A -85,B 0,C 180,E1 6852.55,E2 6852.55} C_VEL
LIN {X 0,Y 627.263,Z 859.31,A -85,B 0,C 180,E1 6858.296,E2 6858.296} C_VEL
LIN {X 0,Y 627.112,Z 859.31,A -85,B 0,C 180,E1 6863.337,E2 6863.337} C_VEL
LIN {X 0,Y 627.053,Z 859.31,A -85,B 0,C 180,E1 6868.891,E2 6868.891} C_VEL
LIN {X 0,Y 626.941,Z 859.31,A -85,B 0,C 180,E1 6874.738,E2 6874.738} C_VEL
LIN {X 0,Y 626.867,Z 859.31,A -85,B 0,C 180,E1 6879.329,E2 6879.329} C_VEL
LIN {X 0,Y 626.809,Z 859.31,A -85,B 0,C 180,E1 6884.495,E2 6884.495} C_VEL
LIN {X 0,Y 626.85,Z 859.31,A -85,B 0,C 180,E1 6889.257,E2 6889.257} C_VEL
LIN {X 0,Y 627.009,Z 859.31,A -85,B 0,C 180,E1 6894.549,E2 6894.549} C_VEL
LIN {X 0,Y 627.048,Z 859.31,A -85,B 0,C 180,E1 6900.19,E2 6900.19} C_VEL
LIN {X 0,Y 643.591,Z 895.521,A -85,B 0,C 180,E1 6901.634,E2 6901.634} C_VEL
LIN {X 0,Y 642.775,Z 969.749,A -85,B 0,C 180,E1 6902.622,E2 6902.622} C_VEL
LIN {X 0,Y 640.961,Z 1007.867,A -85,B 0,C 180,E1 6903.639,E2 6903.639} C_VEL
LIN {X 0,Y 638.436,Z 1044.822,A -85,B 0,C 180,E1 6905.178,E2 6905.178} C_VEL
LIN {X 0,Y 635.554,Z 1080.907,A -85,B 0,C 180,E1 6907.308,E2 6907.308} C_VEL
LIN {X 0,Y 632.823,Z 1112.946,A -85,B 0,C 180,E1 6909.867,E2 6909.867} C_VEL
LIN {X 0,Y 630.655,Z 1141.419,A -85,B 0,C 180,E1 6912.883,E2 6912.883} C_VEL
LIN {X 0,Y 629.08,Z 1165.282,A -85,B 0,C 180,E1 6916.24,E2 6916.24} C_VEL
LIN {X 0,Y 628.323,Z 1182.989,A -85,B 0,C 180,E1 6919.58,E2 6919.58} C_VEL
LIN {X 0,Y 627.918,Z 1195.725,A -85,B 0,C 180,E1 6923.07,E2 6923.07} C_VEL
LIN {X 0,Y 627.847,Z 1202.008,A -85,B 0,C 180,E1 6925.848,E2 6925.848} C_VEL
LIN {X 0,Y 627.762,Z 1205.119,A -85,B 0,C 180,E1 6928.617,E2 6928.617} C_VEL
LIN {X 0,Y 627.829,Z 1205.05,A -85,B 0,C 180,E1 6931.383,E2 6931.383} C_VEL
LIN {X 0,Y 627.944,Z 1200.627,A -85,B 0,C 180,E1 6934.845,E2 6934.845} C_VEL
LIN {X 0,Y 628.129,Z 1190.07,A -85,B 0,C 180,E1 6938.589,E2 6938.589} C_VEL
LIN {X 0,Y 628.709,Z 1173.899,A -85,B 0,C 180,E1 6942.175,E2 6942.175} C_VEL
LIN {X 0,Y 629.787,Z 1152.945,A -85,B 0,C 180,E1 6945.531,E2 6945.531} C_VEL
LIN {X 0,Y 631.607,Z 1127.277,A -85,B 0,C 180,E1 6948.625,E2 6948.625} C_VEL
LIN {X 0,Y 634.123,Z 1097.037,A -85,B 0,C 180,E1 6951.4,E2 6951.4} C_VEL
LIN {X 0,Y 636.87,Z 1064.156,A -85,B 0,C 180,E1 6953.674,E2 6953.674} C_VEL
LIN {X 0,Y 639.543,Z 1029.781,A -85,B 0,C 180,E1 6955.426,E2 6955.426} C_VEL
LIN {X 0,Y 641.727,Z 993.497,A -85,B 0,C 180,E1 6956.715,E2 6956.715} C_VEL
LIN {X 0,Y 643.114,Z 955.727,A -85,B 0,C 180,E1 6957.534,E2 6957.534} C_VEL
LIN {X 0,Y 643.098,Z 894.485,A -85,B 0,C 180,E1 6958.315,E2 6958.315} C_VEL
LIN {X 0,Y 627.043,Z 859.31,A -85,B 0,C 180,E1 6959.769,E2 6959.769} C_VEL
LIN {X 0,Y 627.001,Z 859.31,A -85,B 0,C 180,E1 6965.452,E2 6965.452} C_VEL
LIN {X 0,Y 626.86,Z 859.31,A -85,B 0,C 180,E1 6970.743,E2 6970.743} C_VEL
LIN {X 0,Y 626.813,Z 859.31,A -85,B 0,C 180,E1 6976.489,E2 6976.489} C_VEL
LIN {X 0,Y 626.883,Z 859.31,A -85,B 0,C 180,E1 6981.078,E2 6981.078} C_VEL
LIN {X 0,Y 626.985,Z 859.31,A -85,B 0,C 180,E1 6986.242,E2 6986.242} C_VEL
LIN {X 0,Y 627.043,Z 859.31,A -85,B 0,C 180,E1 6991.109,E2 6991.109} C_VEL
LIN {X 0,Y 627.14,Z 859.31,A -85,B 0,C 180,E1 6996.658,E2 6996.658} C_VEL
LIN {X 0,Y 626.999,Z 859.31,A -85,B 0,C 180,E1 7001.696,E2 7001.696} C_VEL
LIN {X 0,Y 627.283,Z 859.31,A -85,B 0,C 180,E1 7007.449,E2 7007.449} C_VEL
LIN {X 0,Y 627.567,Z 859.31,A -85,B 0,C 180,E1 7013.07,E2 7013.07} C_VEL
LIN {X 0,Y 627.612,Z 859.31,A -85,B 0,C 180,E1 7018.619,E2 7018.619} C_VEL
LIN {X 0,Y 627.599,Z 859.31,A -85,B 0,C 180,E1 7022.769,E2 7022.769} C_VEL
LIN {X 0,Y 627.44,Z 859.31,A -85,B 0,C 180,E1 7028.04,E2 7028.04} C_VEL
LIN {X 0,Y 627.311,Z 859.31,A -85,B 0,C 180,E1 7033.976,E2 7033.976} C_VEL
LIN {X 0,Y 627.312,Z 859.31,A -85,B 0,C 180,E1 7039.599,E2 7039.599} C_VEL
LIN {X 0,Y 627.156,Z 859.31,A -85,B 0,C 180,E1 7044.247,E2 7044.247} C_VEL
LIN {X 0,Y 627.045,Z 859.31,A -85,B 0,C 180,E1 7049.545,E2 7049.545} C_VEL
LIN {X 0,Y 626.948,Z 859.31,A -85,B 0,C 180,E1 7055.447,E2 7055.447} C_VEL
LIN {X 0,Y 626.832,Z 859.31,A -85,B 0,C 180,E1 7060.734,E2 7060.734} C_VEL
LIN {X 0,Y 626.808,Z 859.31,A -85,B 0,C 180,E1 7062.685,E2 7062.685} C_VEL
LIN {X 0,Y 622.831,Z 859.31,A -85,B 0,C 180,E1 7064.251,E2 7064.251} C_VEL
LIN {X 0,Y 618.86,Z 859.31,A -85,B 0,C 180,E1 7065.836,E2 7065.836} C_VEL
LIN {X 0,Y 618.955,Z 859.31,A -85,B 0,C 180,E1 7071.557,E2 7071.557} C_VEL
LIN {X 0,Y 619.145,Z 859.31,A -85,B 0,C 180,E1 7073.317,E2 7073.317} C_VEL
LIN {X 0,Y 638.756,Z 903.855,A -85,B 0,C 180,E1 7074.979,E2 7074.979} C_VEL
LIN {X 0,Y 639.983,Z 909.404,A -85,B 0,C 180,E1 7075.111,E2 7075.111} C_VEL
LIN {X 0,Y 638.385,Z 958.372,A -85,B 0,C 180,E1 7076.007,E2 7076.007} C_VEL
LIN {X 0,Y 636.162,Z 1004.557,A -85,B 0,C 180,E1 7077.465,E2 7077.465} C_VEL
LIN {X 0,Y 633.184,Z 1048.987,A -85,B 0,C 180,E1 7079.508,E2 7079.508} C_VEL
LIN {X 0,Y 630.051,Z 1089.404,A -85,B 0,C 180,E1 7082.032,E2 7082.032} C_VEL
LIN {X 0,Y 627.258,Z 1120.925,A -85,B 0,C 180,E1 7084.616,E2 7084.616} C_VEL
LIN {X 0,Y 624.378,Z 1153.758,A -85,B 0,C 180,E1 7088.091,E2 7088.091} C_VEL
LIN {X 0,Y 622.151,Z 1181.15,A -85,B 0,C 180,E1 7091.845,E2 7091.845} C_VEL
LIN {X 0,Y 620.834,Z 1203.269,A -85,B 0,C 180,E1 7095.873,E2 7095.873} C_VEL
LIN {X 0,Y 620.212,Z 1218.866,A -85,B 0,C 180,E1 7099.797,E2 7099.797} C_VEL
LIN {X 0,Y 619.998,Z 1229.197,A -85,B 0,C 180,E1 7103.686,E2 7103.686} C_VEL
LIN {X 0,Y 619.839,Z 1234.214,A -85,B 0,C 180,E1 7107.197,E2 7107.197} C_VEL
LIN {X 0,Y 619.918,Z 1235.5,A -85,B 0,C 180,E1 7110,E2 7110} C_VEL
LIN {X 0,Y 619.897,Z 1232.649,A -85,B 0,C 180,E1 7114.205,E2 7114.205} C_VEL
LIN {X 0,Y 619.993,Z 1226.126,A -85,B 0,C 180,E1 7117.7,E2 7117.7} C_VEL
LIN {X 0,Y 620.466,Z 1212.934,A -85,B 0,C 180,E1 7121.865,E2 7121.865} C_VEL
LIN {X 0,Y 621.44,Z 1194.756,A -85,B 0,C 180,E1 7125.812,E2 7125.812} C_VEL
LIN {X 0,Y 622.991,Z 1170.532,A -85,B 0,C 180,E1 7129.723,E2 7129.723} C_VEL
LIN {X 0,Y 625.425,Z 1141.652,A -85,B 0,C 180,E1 7133.3,E2 7133.3} C_VEL
LIN {X 0,Y 628.656,Z 1106.042,A -85,B 0,C 180,E1 7136.705,E2 7136.705} C_VEL
LIN {X 0,Y 631.703,Z 1068.985,A -85,B 0,C 180,E1 7139.329,E2 7139.329} C_VEL
LIN {X 0,Y 634.514,Z 1030.068,A -85,B 0,C 180,E1 7141.439,E2 7141.439} C_VEL
LIN {X 0,Y 637.108,Z 986.938,A -85,B 0,C 180,E1 7143.163,E2 7143.163} C_VEL
LIN {X 0,Y 639.149,Z 940.399,A -85,B 0,C 180,E1 7144.392,E2 7144.392} C_VEL
LIN {X 0,Y 639.449,Z 905.043,A -85,B 0,C 180,E1 7144.974,E2 7144.974} C_VEL
LIN {X 0,Y 621.138,Z 865.096,A -85,B 0,C 180,E1 7146.456,E2 7146.456} C_VEL
LIN {X 0,Y 619.127,Z 859.31,A -85,B 0,C 180,E1 7146.681,E2 7146.681} C_VEL
LIN {X 0,Y 619.065,Z 859.31,A -85,B 0,C 180,E1 7152.764,E2 7152.764} C_VEL
LIN {X 0,Y 618.989,Z 859.31,A -85,B 0,C 180,E1 7157.257,E2 7157.257} C_VEL
LIN {X 0,Y 618.933,Z 859.31,A -85,B 0,C 180,E1 7162.271,E2 7162.271} C_VEL
LIN {X 0,Y 619.019,Z 859.31,A -85,B 0,C 180,E1 7167.423,E2 7167.423} C_VEL
LIN {X 0,Y 619.204,Z 859.31,A -85,B 0,C 180,E1 7172.298,E2 7172.298} C_VEL
LIN {X 0,Y 619.277,Z 859.31,A -85,B 0,C 180,E1 7176.957,E2 7176.957} C_VEL
LIN {X 0,Y 619.313,Z 859.31,A -85,B 0,C 180,E1 7182.596,E2 7182.596} C_VEL
LIN {X 0,Y 619.348,Z 859.31,A -85,B 0,C 180,E1 7188.135,E2 7188.135} C_VEL
LIN {X 0,Y 619.626,Z 859.31,A -85,B 0,C 180,E1 7192.977,E2 7192.977} C_VEL
LIN {X 0,Y 619.732,Z 859.31,A -85,B 0,C 180,E1 7198.597,E2 7198.597} C_VEL
LIN {X 0,Y 619.724,Z 859.31,A -85,B 0,C 180,E1 7202.8,E2 7202.8} C_VEL
LIN {X 0,Y 619.528,Z 859.31,A -85,B 0,C 180,E1 7207.021,E2 7207.021} C_VEL
LIN {X 0,Y 619.443,Z 859.31,A -85,B 0,C 180,E1 7212.713,E2 7212.713} C_VEL
LIN {X 0,Y 619.346,Z 859.31,A -85,B 0,C 180,E1 7218.538,E2 7218.538} C_VEL
LIN {X 0,Y 619.211,Z 859.31,A -85,B 0,C 180,E1 7223.042,E2 7223.042} C_VEL
LIN {X 0,Y 619.122,Z 859.31,A -85,B 0,C 180,E1 7228.226,E2 7228.226} C_VEL
LIN {X 0,Y 619.04,Z 859.31,A -85,B 0,C 180,E1 7233.669,E2 7233.669} C_VEL
LIN {X 0,Y 618.942,Z 859.31,A -85,B 0,C 180,E1 7239.519,E2 7239.519} C_VEL
LIN {X 0,Y 618.901,Z 859.31,A -85,B 0,C 180,E1 7245.219,E2 7245.219} C_VEL
LIN {X 0,Y 618.975,Z 859.31,A -85,B 0,C 180,E1 7250.469,E2 7250.469} C_VEL
LIN {X 0,Y 619.077,Z 859.31,A -85,B 0,C 180,E1 7256.3,E2 7256.3} C_VEL
LIN {X 0,Y 619.119,Z 859.818,A -85,B 0,C 180,E1 7259.712,E2 7259.712} C_VEL
LIN {X 0,Y 636.973,Z 897.577,A -85,B 0,C 180,E1 7261.26,E2 7261.26} C_VEL
LIN {X 0,Y 636.25,Z 969.073,A -85,B 0,C 180,E1 7262.207,E2 7262.207} C_VEL
LIN {X 0,Y 634.328,Z 1008.129,A -85,B 0,C 180,E1 7263.246,E2 7263.246} C_VEL
LIN {X 0,Y 631.518,Z 1046.925,A -85,B 0,C 180,E1 7264.887,E2 7264.887} C_VEL
LIN {X 0,Y 628.367,Z 1082.801,A -85,B 0,C 180,E1 7267.069,E2 7267.069} C_VEL
LIN {X 0,Y 625.461,Z 1113.957,A -85,B 0,C 180,E1 7269.619,E2 7269.619} C_VEL
LIN {X 0,Y 623.059,Z 1142.118,A -85,B 0,C 180,E1 7272.667,E2 7272.667} C_VEL
LIN {X 0,Y 621.371,Z 1165.778,A -85,B 0,C 180,E1 7276.066,E2 7276.066} C_VEL
LIN {X 0,Y 620.469,Z 1183.104,A -85,B 0,C 180,E1 7279.446,E2 7279.446} C_VEL
LIN {X 0,Y 620.039,Z 1195.723,A -85,B 0,C 180,E1 7282.981,E2 7282.981} C_VEL
LIN {X 0,Y 619.952,Z 1202.006,A -85,B 0,C 180,E1 7285.795,E2 7285.795} C_VEL
LIN {X 0,Y 619.864,Z 1205.119,A -85,B 0,C 180,E1 7288.599,E2 7288.599} C_VEL
LIN {X 0,Y 619.939,Z 1205.049,A -85,B 0,C 180,E1 7291.401,E2 7291.401} C_VEL
LIN {X 0,Y 620.06,Z 1200.629,A -85,B 0,C 180,E1 7294.907,E2 7294.907} C_VEL
LIN {X 0,Y 620.234,Z 1190.073,A -85,B 0,C 180,E1 7298.7,E2 7298.7} C_VEL
LIN {X 0,Y 620.907,Z 1174.492,A -85,B 0,C 180,E1 7302.286,E2 7302.286} C_VEL
LIN {X 0,Y 622.187,Z 1152.93,A -85,B 0,C 180,E1 7305.814,E2 7305.814} C_VEL
LIN {X 0,Y 624.198,Z 1127.605,A -85,B 0,C 180,E1 7308.919,E2 7308.919} C_VEL
LIN {X 0,Y 626.857,Z 1098.386,A -85,B 0,C 180,E1 7311.648,E2 7311.648} C_VEL
LIN {X 0,Y 629.78,Z 1066.288,A -85,B 0,C 180,E1 7313.932,E2 7313.932} C_VEL
LIN {X 0,Y 632.768,Z 1030.819,A -85,B 0,C 180,E1 7315.78,E2 7315.78} C_VEL
LIN {X 0,Y 635.164,Z 993.477,A -85,B 0,C 180,E1 7317.118,E2 7317.118} C_VEL
LIN {X 0,Y 636.602,Z 955.39,A -85,B 0,C 180,E1 7317.939,E2 7317.939} C_VEL
LIN {X 0,Y 636.478,Z 896.436,A -85,B 0,C 180,E1 7318.691,E2 7318.691} C_VEL
LIN {X 0,Y 619.129,Z 859.31,A -85,B 0,C 180,E1 7320.234,E2 7320.234} C_VEL
LIN {X 0,Y 619.044,Z 859.31,A -85,B 0,C 180,E1 7325.978,E2 7325.978} C_VEL
LIN {X 0,Y 618.928,Z 859.31,A -85,B 0,C 180,E1 7331.379,E2 7331.379} C_VEL
LIN {X 0,Y 618.899,Z 859.31,A -85,B 0,C 180,E1 7337.266,E2 7337.266} C_VEL
LIN {X 0,Y 618.995,Z 859.31,A -85,B 0,C 180,E1 7342.28,E2 7342.28} C_VEL
LIN {X 0,Y 619.033,Z 859.31,A -85,B 0,C 180,E1 7347.429,E2 7347.429} C_VEL
LIN {X 0,Y 619.157,Z 859.31,A -85,B 0,C 180,E1 7352.3,E2 7352.3} C_VEL
LIN {X 0,Y 619.255,Z 859.31,A -85,B 0,C 180,E1 7356.96,E2 7356.96} C_VEL
LIN {X 0,Y 619.088,Z 859.31,A -85,B 0,C 180,E1 7362.664,E2 7362.664} C_VEL
LIN {X 0,Y 619.39,Z 859.31,A -85,B 0,C 180,E1 7368.118,E2 7368.118} C_VEL
LIN {X 0,Y 619.667,Z 859.31,A -85,B 0,C 180,E1 7372.981,E2 7372.981} C_VEL
LIN {X 0,Y 619.735,Z 859.31,A -85,B 0,C 180,E1 7378.601,E2 7378.601} C_VEL
LIN {X 0,Y 619.725,Z 859.31,A -85,B 0,C 180,E1 7382.804,E2 7382.804} C_VEL
LIN {X 0,Y 619.532,Z 859.31,A -85,B 0,C 180,E1 7387.025,E2 7387.025} C_VEL
LIN {X 0,Y 619.423,Z 859.31,A -85,B 0,C 180,E1 7392.717,E2 7392.717} C_VEL
LIN {X 0,Y 619.37,Z 859.31,A -85,B 0,C 180,E1 7398.542,E2 7398.542} C_VEL
LIN {X 0,Y 619.241,Z 859.31,A -85,B 0,C 180,E1 7403.045,E2 7403.045} C_VEL
LIN {X 0,Y 619.148,Z 859.31,A -85,B 0,C 180,E1 7408.229,E2 7408.229} C_VEL
LIN {X 0,Y 619.032,Z 859.31,A -85,B 0,C 180,E1 7413.667,E2 7413.667} C_VEL
LIN {X 0,Y 618.935,Z 859.31,A -85,B 0,C 180,E1 7419.524,E2 7419.524} C_VEL
LIN {X 0,Y 618.916,Z 859.31,A -85,B 0,C 180,E1 7425.223,E2 7425.223} C_VEL
LIN {X 0,Y 618.86,Z 859.31,A -85,B 0,C 180,E1 7425.836,E2 7425.836} C_VEL
LIN {X 0,Y 617.584,Z 859.31,A -85,B 0,C 180,E1 7426.637,E2 7426.637} C_VEL
LIN {X 0,Y 611.009,Z 859.31,A -85,B 0,C 180,E1 7428.814,E2 7428.814} C_VEL
LIN {X 0,Y 610.927,Z 859.31,A -85,B 0,C 180,E1 7429.02,E2 7429.02} C_VEL
LIN {X 0,Y 611.175,Z 859.31,A -85,B 0,C 180,E1 7432.853,E2 7432.853} C_VEL
LIN {X 0,Y 632.957,Z 908.635,A -85,B 0,C 180,E1 7434.757,E2 7434.757} C_VEL
LIN {X 0,Y 631.36,Z 958.102,A -85,B 0,C 180,E1 7435.676,E2 7435.676} C_VEL
LIN {X 0,Y 628.933,Z 1005.782,A -85,B 0,C 180,E1 7437.202,E2 7437.202} C_VEL
LIN {X 0,Y 625.838,Z 1049.989,A -85,B 0,C 180,E1 7439.264,E2 7439.264} C_VEL
LIN {X 0,Y 622.472,Z 1091.178,A -85,B 0,C 180,E1 7441.888,E2 7441.888} C_VEL
LIN {X 0,Y 619.349,Z 1126.402,A -85,B 0,C 180,E1 7444.827,E2 7444.827} C_VEL
LIN {X 0,Y 616.523,Z 1156.708,A -85,B 0,C 180,E1 7448.181,E2 7448.181} C_VEL
LIN {X 0,Y 614.307,Z 1182.936,A -85,B 0,C 180,E1 7451.9,E2 7451.9} C_VEL
LIN {X 0,Y 612.941,Z 1204.99,A -85,B 0,C 180,E1 7456.052,E2 7456.052} C_VEL
LIN {X 0,Y 612.304,Z 1221.162,A -85,B 0,C 180,E1 7460.384,E2 7460.384} C_VEL
LIN {X 0,Y 612.092,Z 1230.458,A -85,B 0,C 180,E1 7464.317,E2 7464.317} C_VEL
LIN {X 0,Y 612.067,Z 1235.166,A -85,B 0,C 180,E1 7468.581,E2 7468.581} C_VEL
LIN {X 0,Y 612.059,Z 1234.214,A -85,B 0,C 180,E1 7472.838,E2 7472.838} C_VEL
LIN {X 0,Y 612.095,Z 1229.199,A -85,B 0,C 180,E1 7476.396,E2 7476.396} C_VEL
LIN {X 0,Y 612.378,Z 1217.719,A -85,B 0,C 180,E1 7480.695,E2 7480.695} C_VEL
LIN {X 0,Y 613.138,Z 1201.689,A -85,B 0,C 180,E1 7484.64,E2 7484.64} C_VEL
LIN {X 0,Y 614.497,Z 1180.337,A -85,B 0,C 180,E1 7488.514,E2 7488.514} C_VEL
LIN {X 0,Y 616.93,Z 1152.433,A -85,B 0,C 180,E1 7492.356,E2 7492.356} C_VEL
LIN {X 0,Y 619.888,Z 1120.833,A -85,B 0,C 180,E1 7495.691,E2 7495.691} C_VEL
LIN {X 0,Y 622.991,Z 1084.95,A -85,B 0,C 180,E1 7498.551,E2 7498.551} C_VEL
LIN {X 0,Y 626.119,Z 1046.073,A -85,B 0,C 180,E1 7500.941,E2 7500.941} C_VEL
LIN {X 0,Y 629.073,Z 1005.08,A -85,B 0,C 180,E1 7502.821,E2 7502.821} C_VEL
LIN {X 0,Y 631.486,Z 959.665,A -85,B 0,C 180,E1 7504.272,E2 7504.272} C_VEL
LIN {X 0,Y 632.951,Z 914.463,A -85,B 0,C 180,E1 7505.154,E2 7505.154} C_VEL
LIN {X 0,Y 632.319,Z 907.272,A -85,B 0,C 180,E1 7505.292,E2 7505.292} C_VEL
LIN {X 0,Y 611.255,Z 860.267,A -85,B 0,C 180,E1 7507.111,E2 7507.111} C_VEL
LIN {X 0,Y 611.166,Z 859.31,A -85,B 0,C 180,E1 7507.146,E2 7507.146} C_VEL
LIN {X 0,Y 611.092,Z 859.31,A -85,B 0,C 180,E1 7512.029,E2 7512.029} C_VEL
LIN {X 0,Y 611.059,Z 859.31,A -85,B 0,C 180,E1 7517.98,E2 7517.98} C_VEL
LIN {X 0,Y 611,Z 859.31,A -85,B 0,C 180,E1 7523.482,E2 7523.482} C_VEL
LIN {X 0,Y 611.125,Z 859.31,A -85,B 0,C 180,E1 7528.628,E2 7528.628} C_VEL
LIN {X 0,Y 611.308,Z 859.31,A -85,B 0,C 180,E1 7533.507,E2 7533.507} C_VEL
LIN {X 0,Y 611.37,Z 859.31,A -85,B 0,C 180,E1 7538.179,E2 7538.179} C_VEL
LIN {X 0,Y 611.433,Z 859.31,A -85,B 0,C 180,E1 7542.702,E2 7542.702} C_VEL
LIN {X 0,Y 611.521,Z 859.31,A -85,B 0,C 180,E1 7548.567,E2 7548.567} C_VEL
LIN {X 0,Y 611.715,Z 859.31,A -85,B 0,C 180,E1 7554.313,E2 7554.313} C_VEL
LIN {X 0,Y 611.832,Z 859.31,A -85,B 0,C 180,E1 7558.579,E2 7558.579} C_VEL
LIN {X 0,Y 611.821,Z 859.31,A -85,B 0,C 180,E1 7562.837,E2 7562.837} C_VEL
LIN {X 0,Y 611.581,Z 859.31,A -85,B 0,C 180,E1 7567.666,E2 7567.666} C_VEL
LIN {X 0,Y 611.522,Z 859.31,A -85,B 0,C 180,E1 7572.88,E2 7572.88} C_VEL
LIN {X 0,Y 611.473,Z 859.31,A -85,B 0,C 180,E1 7577.293,E2 7577.293} C_VEL
LIN {X 0,Y 611.346,Z 859.31,A -85,B 0,C 180,E1 7581.818,E2 7581.818} C_VEL
LIN {X 0,Y 611.21,Z 859.31,A -85,B 0,C 180,E1 7586.811,E2 7586.811} C_VEL
LIN {X 0,Y 611.135,Z 859.31,A -85,B 0,C 180,E1 7592.54,E2 7592.54} C_VEL
LIN {X 0,Y 611.031,Z 859.31,A -85,B 0,C 180,E1 7598.3,E2 7598.3} C_VEL
LIN {X 0,Y 610.967,Z 859.31,A -85,B 0,C 180,E1 7604.008,E2 7604.008} C_VEL
LIN {X 0,Y 611.07,Z 859.31,A -85,B 0,C 180,E1 7610.218,E2 7610.218} C_VEL
LIN {X 0,Y 611.107,Z 859.31,A -85,B 0,C 180,E1 7615.229,E2 7615.229} C_VEL
LIN {X 0,Y 611.144,Z 859.679,A -85,B 0,C 180,E1 7619.204,E2 7619.204} C_VEL
LIN {X 0,Y 630.456,Z 899.866,A -85,B 0,C 180,E1 7620.897,E2 7620.897} C_VEL
LIN {X 0,Y 629.642,Z 969.789,A -85,B 0,C 180,E1 7621.825,E2 7621.825} C_VEL
LIN {X 0,Y 627.604,Z 1009.767,A -85,B 0,C 180,E1 7622.901,E2 7622.901} C_VEL
LIN {X 0,Y 624.756,Z 1047.184,A -85,B 0,C 180,E1 7624.5,E2 7624.5} C_VEL
LIN {X 0,Y 621.432,Z 1082.509,A -85,B 0,C 180,E1 7626.66,E2 7626.66} C_VEL
LIN {X 0,Y 618.096,Z 1115.004,A -85,B 0,C 180,E1 7629.365,E2 7629.365} C_VEL
LIN {X 0,Y 615.5,Z 1142.884,A -85,B 0,C 180,E1 7632.448,E2 7632.448} C_VEL
LIN {X 0,Y 613.718,Z 1165.241,A -85,B 0,C 180,E1 7635.706,E2 7635.706} C_VEL
LIN {X 0,Y 612.662,Z 1183.474,A -85,B 0,C 180,E1 7639.31,E2 7639.31} C_VEL
LIN {X 0,Y 612.166,Z 1195.891,A -85,B 0,C 180,E1 7642.891,E2 7642.891} C_VEL
LIN {X 0,Y 612.059,Z 1202.064,A -85,B 0,C 180,E1 7645.741,E2 7645.741} C_VEL
LIN {X 0,Y 611.964,Z 1205.134,A -85,B 0,C 180,E1 7648.581,E2 7648.581} C_VEL
LIN {X 0,Y 612.038,Z 1205.064,A -85,B 0,C 180,E1 7651.419,E2 7651.419} C_VEL
LIN {X 0,Y 612.187,Z 1200.709,A -85,B 0,C 180,E1 7654.97,E2 7654.97} C_VEL
LIN {X 0,Y 612.382,Z 1190.079,A -85,B 0,C 180,E1 7658.897,E2 7658.897} C_VEL
LIN {X 0,Y 613.16,Z 1173.941,A -85,B 0,C 180,E1 7662.636,E2 7662.636} C_VEL
LIN {X 0,Y 614.64,Z 1152.68,A -85,B 0,C 180,E1 7666.148,E2 7666.148} C_VEL
LIN {X 0,Y 616.923,Z 1127.102,A -85,B 0,C 180,E1 7669.307,E2 7669.307} C_VEL
LIN {X 0,Y 619.93,Z 1096.634,A -85,B 0,C 180,E1 7672.168,E2 7672.168} C_VEL
LIN {X 0,Y 623.24,Z 1063.26,A -85,B 0,C 180,E1 7674.51,E2 7674.51} C_VEL
LIN {X 0,Y 626.23,Z 1029.01,A -85,B 0,C 180,E1 7676.259,E2 7676.259} C_VEL
LIN {X 0,Y 628.566,Z 991.987,A -85,B 0,C 180,E1 7677.56,E2 7677.56} C_VEL
LIN {X 0,Y 630.012,Z 954.8,A -85,B 0,C 180,E1 7678.343,E2 7678.343} C_VEL
LIN {X 0,Y 629.952,Z 898.664,A -85,B 0,C 180,E1 7679.056,E2 7679.056} C_VEL
LIN {X 0,Y 611.205,Z 859.31,A -85,B 0,C 180,E1 7680.745,E2 7680.745} C_VEL
LIN {X 0,Y 611.088,Z 859.31,A -85,B 0,C 180,E1 7686.521,E2 7686.521} C_VEL
LIN {X 0,Y 610.983,Z 859.31,A -85,B 0,C 180,E1 7692.038,E2 7692.038} C_VEL
LIN {X 0,Y 610.971,Z 859.31,A -85,B 0,C 180,E1 7698.077,E2 7698.077} C_VEL
LIN {X 0,Y 611.094,Z 859.31,A -85,B 0,C 180,E1 7703.493,E2 7703.493} C_VEL
LIN {X 0,Y 611.106,Z 859.31,A -85,B 0,C 180,E1 7708.631,E2 7708.631} C_VEL
LIN {X 0,Y 611.251,Z 859.31,A -85,B 0,C 180,E1 7713.508,E2 7713.508} C_VEL
LIN {X 0,Y 611.356,Z 859.31,A -85,B 0,C 180,E1 7718.182,E2 7718.182} C_VEL
LIN {X 0,Y 611.231,Z 859.31,A -85,B 0,C 180,E1 7724.181,E2 7724.181} C_VEL
LIN {X 0,Y 611.553,Z 859.31,A -85,B 0,C 180,E1 7728.572,E2 7728.572} C_VEL
LIN {X 0,Y 611.751,Z 859.31,A -85,B 0,C 180,E1 7732.89,E2 7732.89} C_VEL
LIN {X 0,Y 611.835,Z 859.31,A -85,B 0,C 180,E1 7738.583,E2 7738.583} C_VEL
LIN {X 0,Y 611.822,Z 859.31,A -85,B 0,C 180,E1 7742.84,E2 7742.84} C_VEL
LIN {X 0,Y 611.588,Z 859.31,A -85,B 0,C 180,E1 7747.668,E2 7747.668} C_VEL
LIN {X 0,Y 611.503,Z 859.31,A -85,B 0,C 180,E1 7752.885,E2 7752.885} C_VEL
LIN {X 0,Y 611.479,Z 859.31,A -85,B 0,C 180,E1 7757.297,E2 7757.297} C_VEL
LIN {X 0,Y 611.367,Z 859.31,A -85,B 0,C 180,E1 7761.821,E2 7761.821} C_VEL
LIN {X 0,Y 611.253,Z 859.31,A -85,B 0,C 180,E1 7766.818,E2 7766.818} C_VEL
LIN {X 0,Y 611.137,Z 859.31,A -85,B 0,C 180,E1 7772.539,E2 7772.539} C_VEL
LIN {X 0,Y 611.031,Z 859.31,A -85,B 0,C 180,E1 7778.305,E2 7778.305} C_VEL
LIN {X 0,Y 610.97,Z 859.31,A -85,B 0,C 180,E1 7784.008,E2 7784.008} C_VEL
LIN {X 0,Y 610.927,Z 859.31,A -85,B 0,C 180,E1 7789.02,E2 7789.02} C_VEL
LIN {X 0,Y 609.701,Z 859.31,A -85,B 0,C 180,E1 7789.834,E2 7789.834} C_VEL
LIN {X 0,Y 603.25,Z 859.31,A -85,B 0,C 180,E1 7792.048,E2 7792.048} C_VEL
LIN {X 0,Y 603.19,Z 859.31,A -85,B 0,C 180,E1 7792.258,E2 7792.258} C_VEL
LIN {X 0,Y 603.616,Z 861.777,A -85,B 0,C 180,E1 7792.438,E2 7792.438} C_VEL
LIN {X 0,Y 626.008,Z 911.119,A -85,B 0,C 180,E1 7794.45,E2 7794.45} C_VEL
LIN {X 0,Y 624.328,Z 958.338,A -85,B 0,C 180,E1 7795.352,E2 7795.352} C_VEL
LIN {X 0,Y 621.775,Z 1004.45,A -85,B 0,C 180,E1 7796.835,E2 7796.835} C_VEL
LIN {X 0,Y 618.557,Z 1049.614,A -85,B 0,C 180,E1 7798.948,E2 7798.948} C_VEL
LIN {X 0,Y 615.136,Z 1089.371,A -85,B 0,C 180,E1 7801.482,E2 7801.482} C_VEL
LIN {X 0,Y 611.995,Z 1124.244,A -85,B 0,C 180,E1 7804.382,E2 7804.382} C_VEL
LIN {X 0,Y 609.332,Z 1153.194,A -85,B 0,C 180,E1 7807.446,E2 7807.446} C_VEL
LIN {X 0,Y 606.768,Z 1181.37,A -85,B 0,C 180,E1 7811.403,E2 7811.403} C_VEL
LIN {X 0,Y 605.22,Z 1203.267,A -85,B 0,C 180,E1 7815.5,E2 7815.5} C_VEL
LIN {X 0,Y 604.516,Z 1218.866,A -85,B 0,C 180,E1 7819.529,E2 7819.529} C_VEL
LIN {X 0,Y 604.22,Z 1229.198,A -85,B 0,C 180,E1 7823.52,E2 7823.52} C_VEL
LIN {X 0,Y 604.05,Z 1234.213,A -85,B 0,C 180,E1 7827.124,E2 7827.124} C_VEL
LIN {X 0,Y 604.13,Z 1235.5,A -85,B 0,C 180,E1 7830,E2 7830} C_VEL
LIN {X 0,Y 604.109,Z 1232.648,A -85,B 0,C 180,E1 7834.315,E2 7834.315} C_VEL
LIN {X 0,Y 604.241,Z 1225.75,A -85,B 0,C 180,E1 7838.055,E2 7838.055} C_VEL
LIN {X 0,Y 604.818,Z 1212.309,A -85,B 0,C 180,E1 7842.348,E2 7842.348} C_VEL
LIN {X 0,Y 605.865,Z 1194.166,A -85,B 0,C 180,E1 7846.342,E2 7846.342} C_VEL
LIN {X 0,Y 607.661,Z 1170.529,A -85,B 0,C 180,E1 7850.242,E2 7850.242} C_VEL
LIN {X 0,Y 610.383,Z 1142.419,A -85,B 0,C 180,E1 7853.791,E2 7853.791} C_VEL
LIN {X 0,Y 613.453,Z 1108.376,A -85,B 0,C 180,E1 7857.028,E2 7857.028} C_VEL
LIN {X 0,Y 616.759,Z 1071.601,A -85,B 0,C 180,E1 7859.734,E2 7859.734} C_VEL
LIN {X 0,Y 619.934,Z 1031.859,A -85,B 0,C 180,E1 7861.961,E2 7861.961} C_VEL
LIN {X 0,Y 622.841,Z 987.072,A -85,B 0,C 180,E1 7863.794,E2 7863.794} C_VEL
LIN {X 0,Y 625.167,Z 939.357,A -85,B 0,C 180,E1 7865.079,E2 7865.079} C_VEL
LIN {X 0,Y 625.449,Z 910.09,A -85,B 0,C 180,E1 7865.594,E2 7865.594} C_VEL
LIN {X 0,Y 603.204,Z 859.31,A -85,B 0,C 180,E1 7867.659,E2 7867.659} C_VEL
LIN {X 0,Y 603.156,Z 859.31,A -85,B 0,C 180,E1 7873.248,E2 7873.248} C_VEL
LIN {X 0,Y 603.087,Z 859.31,A -85,B 0,C 180,E1 7879.222,E2 7879.222} C_VEL
LIN {X 0,Y 603.096,Z 859.31,A -85,B 0,C 180,E1 7884.707,E2 7884.707} C_VEL
LIN {X 0,Y 603.248,Z 859.31,A -85,B 0,C 180,E1 7889.849,E2 7889.849} C_VEL
LIN {X 0,Y 603.422,Z 859.31,A -85,B 0,C 180,E1 7894.734,E2 7894.734} C_VEL
LIN {X 0,Y 603.463,Z 859.31,A -85,B 0,C 180,E1 7899.422,E2 7899.422} C_VEL
LIN {X 0,Y 603.51,Z 859.31,A -85,B 0,C 180,E1 7903.97,E2 7903.97} C_VEL
LIN {X 0,Y 603.628,Z 859.31,A -85,B 0,C 180,E1 7909.88,E2 7909.88} C_VEL
LIN {X 0,Y 603.832,Z 859.31,A -85,B 0,C 180,E1 7914.239,E2 7914.239} C_VEL
LIN {X 0,Y 603.933,Z 859.31,A -85,B 0,C 180,E1 7918.561,E2 7918.561} C_VEL
LIN {X 0,Y 603.927,Z 859.31,A -85,B 0,C 180,E1 7922.874,E2 7922.874} C_VEL
LIN {X 0,Y 603.71,Z 859.31,A -85,B 0,C 180,E1 7927.206,E2 7927.206} C_VEL
LIN {X 0,Y 603.602,Z 859.31,A -85,B 0,C 180,E1 7933.052,E2 7933.052} C_VEL
LIN {X 0,Y 603.55,Z 859.31,A -85,B 0,C 180,E1 7937.527,E2 7937.527} C_VEL
LIN {X 0,Y 603.42,Z 859.31,A -85,B 0,C 180,E1 7942.12,E2 7942.12} C_VEL
LIN {X 0,Y 603.329,Z 859.31,A -85,B 0,C 180,E1 7946.867,E2 7946.867} C_VEL
LIN {X 0,Y 603.224,Z 859.31,A -85,B 0,C 180,E1 7951.826,E2 7951.826} C_VEL
LIN {X 0,Y 603.118,Z 859.31,A -85,B 0,C 180,E1 7957.07,E2 7957.07} C_VEL
LIN {X 0,Y 603.001,Z 859.31,A -85,B 0,C 180,E1 7962.709,E2 7962.709} C_VEL
LIN {X 0,Y 602.993,Z 859.31,A -85,B 0,C 180,E1 7967.274,E2 7967.274} C_VEL
LIN {X 0,Y 603.168,Z 859.31,A -85,B 0,C 180,E1 7972.92,E2 7972.92} C_VEL
LIN {X 0,Y 603.214,Z 859.31,A -85,B 0,C 180,E1 7978.659,E2 7978.659} C_VEL
LIN {X 0,Y 624.001,Z 904.223,A -85,B 0,C 180,E1 7980.56,E2 7980.56} C_VEL
LIN {X 0,Y 622.966,Z 970.998,A -85,B 0,C 180,E1 7981.452,E2 7981.452} C_VEL
LIN {X 0,Y 620.763,Z 1011.528,A -85,B 0,C 180,E1 7982.57,E2 7982.57} C_VEL
LIN {X 0,Y 617.803,Z 1048.768,A -85,B 0,C 180,E1 7984.192,E2 7984.192} C_VEL
LIN {X 0,Y 614.401,Z 1083.156,A -85,B 0,C 180,E1 7986.314,E2 7986.314} C_VEL
LIN {X 0,Y 610.853,Z 1115.056,A -85,B 0,C 180,E1 7988.997,E2 7988.997} C_VEL
LIN {X 0,Y 608.066,Z 1142.274,A -85,B 0,C 180,E1 7992.038,E2 7992.038} C_VEL
LIN {X 0,Y 605.996,Z 1165.808,A -85,B 0,C 180,E1 7995.52,E2 7995.52} C_VEL
LIN {X 0,Y 604.83,Z 1183.858,A -85,B 0,C 180,E1 7999.17,E2 7999.17} C_VEL
LIN {X 0,Y 604.305,Z 1196.17,A -85,B 0,C 180,E1 8002.798,E2 8002.798} C_VEL
LIN {X 0,Y 604.194,Z 1202.292,A -85,B 0,C 180,E1 8005.685,E2 8005.685} C_VEL
LIN {X 0,Y 604.066,Z 1205.339,A -85,B 0,C 180,E1 8008.563,E2 8008.563} C_VEL
LIN {X 0,Y 604.164,Z 1205.272,A -85,B 0,C 180,E1 8011.437,E2 8011.437} C_VEL
LIN {X 0,Y 604.291,Z 1200.952,A -85,B 0,C 180,E1 8015.035,E2 8015.035} C_VEL
LIN {X 0,Y 604.513,Z 1190.411,A -85,B 0,C 180,E1 8019.014,E2 8019.014} C_VEL
LIN {X 0,Y 605.372,Z 1174.853,A -85,B 0,C 180,E1 8022.721,E2 8022.721} C_VEL
LIN {X 0,Y 606.915,Z 1154.577,A -85,B 0,C 180,E1 8026.182,E2 8026.182} C_VEL
LIN {X 0,Y 609.361,Z 1129.445,A -85,B 0,C 180,E1 8029.407,E2 8029.407} C_VEL
LIN {X 0,Y 612.516,Z 1100.152,A -85,B 0,C 180,E1 8032.26,E2 8032.26} C_VEL
LIN {X 0,Y 615.944,Z 1067.472,A -85,B 0,C 180,E1 8034.646,E2 8034.646} C_VEL
LIN {X 0,Y 619.207,Z 1032.107,A -85,B 0,C 180,E1 8036.516,E2 8036.516} C_VEL
LIN {X 0,Y 621.775,Z 994.939,A -85,B 0,C 180,E1 8037.869,E2 8037.869} C_VEL
LIN {X 0,Y 623.392,Z 955.25,A -85,B 0,C 180,E1 8038.733,E2 8038.733} C_VEL
LIN {X 0,Y 623.24,Z 900.996,A -85,B 0,C 180,E1 8039.433,E2 8039.433} C_VEL
LIN {X 0,Y 603.488,Z 861.247,A -85,B 0,C 180,E1 8041.182,E2 8041.182} C_VEL
LIN {X 0,Y 603.252,Z 859.31,A -85,B 0,C 180,E1 8041.318,E2 8041.318} C_VEL
LIN {X 0,Y 603.167,Z 859.31,A -85,B 0,C 180,E1 8047.081,E2 8047.081} C_VEL
LIN {X 0,Y 602.997,Z 859.31,A -85,B 0,C 180,E1 8052.726,E2 8052.726} C_VEL
LIN {X 0,Y 602.986,Z 859.31,A -85,B 0,C 180,E1 8057.29,E2 8057.29} C_VEL
LIN {X 0,Y 603.165,Z 859.31,A -85,B 0,C 180,E1 8062.933,E2 8062.933} C_VEL
LIN {X 0,Y 603.232,Z 859.31,A -85,B 0,C 180,E1 8068.657,E2 8068.657} C_VEL
LIN {X 0,Y 603.344,Z 859.31,A -85,B 0,C 180,E1 8073.133,E2 8073.133} C_VEL
LIN {X 0,Y 603.46,Z 859.31,A -85,B 0,C 180,E1 8078.291,E2 8078.291} C_VEL
LIN {X 0,Y 603.3,Z 859.31,A -85,B 0,C 180,E1 8083.968,E2 8083.968} C_VEL
LIN {X 0,Y 603.621,Z 859.31,A -85,B 0,C 180,E1 8088.42,E2 8088.42} C_VEL
LIN {X 0,Y 603.855,Z 859.31,A -85,B 0,C 180,E1 8092.796,E2 8092.796} C_VEL
LIN {X 0,Y 603.936,Z 859.31,A -85,B 0,C 180,E1 8098.565,E2 8098.565} C_VEL
LIN {X 0,Y 603.928,Z 859.31,A -85,B 0,C 180,E1 8102.878,E2 8102.878} C_VEL
LIN {X 0,Y 603.714,Z 859.31,A -85,B 0,C 180,E1 8107.21,E2 8107.21} C_VEL
LIN {X 0,Y 603.588,Z 859.31,A -85,B 0,C 180,E1 8113.057,E2 8113.057} C_VEL
LIN {X 0,Y 603.563,Z 859.31,A -85,B 0,C 180,E1 8117.531,E2 8117.531} C_VEL
LIN {X 0,Y 603.442,Z 859.31,A -85,B 0,C 180,E1 8122.123,E2 8122.123} C_VEL
LIN {X 0,Y 603.371,Z 859.31,A -85,B 0,C 180,E1 8126.87,E2 8126.87} C_VEL
LIN {X 0,Y 603.232,Z 859.31,A -85,B 0,C 180,E1 8131.83,E2 8131.83} C_VEL
LIN {X 0,Y 603.123,Z 859.31,A -85,B 0,C 180,E1 8137.074,E2 8137.074} C_VEL
LIN {X 0,Y 603.009,Z 859.31,A -85,B 0,C 180,E1 8143.219,E2 8143.219} C_VEL
LIN {X 0,Y 603.04,Z 859.31,A -85,B 0,C 180,E1 8149.208,E2 8149.208} C_VEL
LIN {X 0,Y 603.19,Z 859.31,A -85,B 0,C 180,E1 8152.258,E2 8152.258} C_VEL
LIN {X 0,Y 605.665,Z 862.192,A -85,B 0,C 180,E1 8152.573,E2 8152.573} C_VEL
LIN {X 0,Y 608.163,Z 873.214,A -85,B 0,C 180,E1 8152.874,E2 8152.874} C_VEL
LIN {X 0,Y 609.11,Z 891.12,A -85,B 0,C 180,E1 8153.212,E2 8153.212} C_VEL
LIN {X 0,Y 609.481,Z 892.287,A -85,B 0,C 180,E1 8153.253,E2 8153.253} C_VEL
LIN {X 0,Y 619.106,Z 915.144,A -85,B 0,C 180,E1 8154.151,E2 8154.151} C_VEL
LIN {X 0,Y 617.093,Z 961.55,A -85,B 0,C 180,E1 8155.099,E2 8155.099} C_VEL
LIN {X 0,Y 614.524,Z 1006.962,A -85,B 0,C 180,E1 8156.621,E2 8156.621} C_VEL
LIN {X 0,Y 611.112,Z 1051.281,A -85,B 0,C 180,E1 8158.746,E2 8158.746} C_VEL
LIN {X 0,Y 607.475,Z 1092.401,A -85,B 0,C 180,E1 8161.422,E2 8161.422} C_VEL
LIN {X 0,Y 603.93,Z 1129.724,A -85,B 0,C 180,E1 8164.656,E2 8164.656} C_VEL
LIN {X 0,Y 600.881,Z 1161.855,A -85,B 0,C 180,E1 8168.301,E2 8168.301} C_VEL
LIN {X 0,Y 598.648,Z 1185.754,A -85,B 0,C 180,E1 8171.905,E2 8171.905} C_VEL
LIN {X 0,Y 597.317,Z 1204.991,A -85,B 0,C 180,E1 8175.68,E2 8175.68} C_VEL
LIN {X 0,Y 596.568,Z 1220.014,A -85,B 0,C 180,E1 8179.758,E2 8179.758} C_VEL
LIN {X 0,Y 596.34,Z 1229.198,A -85,B 0,C 180,E1 8183.434,E2 8183.434} C_VEL
LIN {X 0,Y 596.147,Z 1234.212,A -85,B 0,C 180,E1 8187.086,E2 8187.086} C_VEL
LIN {X 0,Y 596.23,Z 1235.5,A -85,B 0,C 180,E1 8190,E2 8190} C_VEL
LIN {X 0,Y 596.215,Z 1232.647,A -85,B 0,C 180,E1 8194.373,E2 8194.373} C_VEL
LIN {X 0,Y 596.361,Z 1225.735,A -85,B 0,C 180,E1 8198.168,E2 8198.168} C_VEL
LIN {X 0,Y 596.969,Z 1212.309,A -85,B 0,C 180,E1 8202.513,E2 8202.513} C_VEL
LIN {X 0,Y 598.062,Z 1194.165,A -85,B 0,C 180,E1 8206.561,E2 8206.561} C_VEL
LIN {X 0,Y 599.985,Z 1170.526,A -85,B 0,C 180,E1 8210.513,E2 8210.513} C_VEL
LIN {X 0,Y 602.781,Z 1141.599,A -85,B 0,C 180,E1 8214.11,E2 8214.11} C_VEL
LIN {X 0,Y 606.28,Z 1105.419,A -85,B 0,C 180,E1 8217.548,E2 8217.548} C_VEL
LIN {X 0,Y 609.893,Z 1066.129,A -85,B 0,C 180,E1 8220.371,E2 8220.371} C_VEL
LIN {X 0,Y 613.381,Z 1023.563,A -85,B 0,C 180,E1 8222.658,E2 8222.658} C_VEL
LIN {X 0,Y 616.181,Z 980.374,A -85,B 0,C 180,E1 8224.338,E2 8224.338} C_VEL
LIN {X 0,Y 618.392,Z 934.594,A -85,B 0,C 180,E1 8225.521,E2 8225.521} C_VEL
LIN {X 0,Y 618.526,Z 912.514,A -85,B 0,C 180,E1 8225.924,E2 8225.924} C_VEL
LIN {X 0,Y 595.266,Z 859.31,A -85,B 0,C 180,E1 8228.217,E2 8228.217} C_VEL
LIN {X 0,Y 595.249,Z 859.31,A -85,B 0,C 180,E1 8233.418,E2 8233.418} C_VEL
LIN {X 0,Y 595.159,Z 859.31,A -85,B 0,C 180,E1 8238.561,E2 8238.561} C_VEL
LIN {X 0,Y 595.205,Z 859.31,A -85,B 0,C 180,E1 8244.554,E2 8244.554} C_VEL
LIN {X 0,Y 595.369,Z 859.31,A -85,B 0,C 180,E1 8249.922,E2 8249.922} C_VEL
LIN {X 0,Y 595.498,Z 859.31,A -85,B 0,C 180,E1 8254.374,E2 8254.374} C_VEL
LIN {X 0,Y 595.535,Z 859.31,A -85,B 0,C 180,E1 8260.294,E2 8260.294} C_VEL
LIN {X 0,Y 595.608,Z 859.31,A -85,B 0,C 180,E1 8265.263,E2 8265.263} C_VEL
LIN {X 0,Y 595.801,Z 859.31,A -85,B 0,C 180,E1 8271.223,E2 8271.223} C_VEL
LIN {X 0,Y 596.084,Z 859.31,A -85,B 0,C 180,E1 8277.085,E2 8277.085} C_VEL
LIN {X 0,Y 596.197,Z 859.31,A -85,B 0,C 180,E1 8281.454,E2 8281.454} C_VEL
LIN {X 0,Y 595.976,Z 859.31,A -85,B 0,C 180,E1 8285.834,E2 8285.834} C_VEL
LIN {X 0,Y 595.753,Z 859.31,A -85,B 0,C 180,E1 8291.735,E2 8291.735} C_VEL
LIN {X 0,Y 595.633,Z 859.31,A -85,B 0,C 180,E1 8296.244,E2 8296.244} C_VEL
LIN {X 0,Y 595.533,Z 859.31,A -85,B 0,C 180,E1 8300.86,E2 8300.86} C_VEL
LIN {X 0,Y 595.403,Z 859.31,A -85,B 0,C 180,E1 8305.626,E2 8305.626} C_VEL
LIN {X 0,Y 595.308,Z 859.31,A -85,B 0,C 180,E1 8310.591,E2 8310.591} C_VEL
LIN {X 0,Y 595.218,Z 859.31,A -85,B 0,C 180,E1 8315.827,E2 8315.827} C_VEL
LIN {X 0,Y 595.098,Z 859.31,A -85,B 0,C 180,E1 8321.439,E2 8321.439} C_VEL
LIN {X 0,Y 595.102,Z 859.31,A -85,B 0,C 180,E1 8326.568,E2 8326.568} C_VEL
LIN {X 0,Y 595.194,Z 859.31,A -85,B 0,C 180,E1 8332.338,E2 8332.338} C_VEL
LIN {X 0,Y 595.311,Z 859.31,A -85,B 0,C 180,E1 8338.138,E2 8338.138} C_VEL
LIN {X 0,Y 605.885,Z 881.805,A -85,B 0,C 180,E1 8339.142,E2 8339.142} C_VEL
LIN {X 0,Y 617.239,Z 904.739,A -85,B 0,C 180,E1 8340.151,E2 8340.151} C_VEL
LIN {X 0,Y 616.289,Z 971.799,A -85,B 0,C 180,E1 8341.069,E2 8341.069} C_VEL
LIN {X 0,Y 613.963,Z 1012.142,A -85,B 0,C 180,E1 8342.2,E2 8342.2} C_VEL
LIN {X 0,Y 610.809,Z 1049.984,A -85,B 0,C 180,E1 8343.875,E2 8343.875} C_VEL
LIN {X 0,Y 607.265,Z 1084.056,A -85,B 0,C 180,E1 8346.002,E2 8346.002} C_VEL
LIN {X 0,Y 603.567,Z 1115.947,A -85,B 0,C 180,E1 8348.709,E2 8348.709} C_VEL
LIN {X 0,Y 600.544,Z 1143.276,A -85,B 0,C 180,E1 8351.827,E2 8351.827} C_VEL
LIN {X 0,Y 598.303,Z 1166.386,A -85,B 0,C 180,E1 8355.329,E2 8355.329} C_VEL
LIN {X 0,Y 597.018,Z 1184.262,A -85,B 0,C 180,E1 8359.027,E2 8359.027} C_VEL
LIN {X 0,Y 596.443,Z 1196.452,A -85,B 0,C 180,E1 8362.702,E2 8362.702} C_VEL
LIN {X 0,Y 596.305,Z 1202.525,A -85,B 0,C 180,E1 8365.628,E2 8365.628} C_VEL
LIN {X 0,Y 596.169,Z 1205.545,A -85,B 0,C 180,E1 8368.544,E2 8368.544} C_VEL
LIN {X 0,Y 596.265,Z 1205.48,A -85,B 0,C 180,E1 8371.456,E2 8371.456} C_VEL
LIN {X 0,Y 596.395,Z 1201.196,A -85,B 0,C 180,E1 8375.102,E2 8375.102} C_VEL
LIN {X 0,Y 596.666,Z 1190.771,A -85,B 0,C 180,E1 8379.133,E2 8379.133} C_VEL
LIN {X 0,Y 597.633,Z 1174.901,A -85,B 0,C 180,E1 8382.979,E2 8382.979} C_VEL
LIN {X 0,Y 599.378,Z 1154.44,A -85,B 0,C 180,E1 8386.524,E2 8386.524} C_VEL
LIN {X 0,Y 602.139,Z 1128.622,A -85,B 0,C 180,E1 8389.861,E2 8389.861} C_VEL
LIN {X 0,Y 605.417,Z 1100.24,A -85,B 0,C 180,E1 8392.633,E2 8392.633} C_VEL
LIN {X 0,Y 608.964,Z 1067.514,A -85,B 0,C 180,E1 8395.025,E2 8395.025} C_VEL
LIN {X 0,Y 612.424,Z 1031.879,A -85,B 0,C 180,E1 8396.914,E2 8396.914} C_VEL
LIN {X 0,Y 615.064,Z 994.703,A -85,B 0,C 180,E1 8398.273,E2 8398.273} C_VEL
LIN {X 0,Y 616.796,Z 955.16,A -85,B 0,C 180,E1 8399.134,E2 8399.134} C_VEL
LIN {X 0,Y 616.842,Z 903.92,A -85,B 0,C 180,E1 8399.792,E2 8399.792} C_VEL
LIN {X 0,Y 595.45,Z 860.429,A -85,B 0,C 180,E1 8401.733,E2 8401.733} C_VEL
LIN {X 0,Y 595.36,Z 859.31,A -85,B 0,C 180,E1 8401.875,E2 8401.875} C_VEL
LIN {X 0,Y 595.196,Z 859.31,A -85,B 0,C 180,E1 8407.663,E2 8407.663} C_VEL
LIN {X 0,Y 595.105,Z 859.31,A -85,B 0,C 180,E1 8413.432,E2 8413.432} C_VEL
LIN {X 0,Y 595.093,Z 859.31,A -85,B 0,C 180,E1 8418.56,E2 8418.56} C_VEL
LIN {X 0,Y 595.276,Z 859.31,A -85,B 0,C 180,E1 8424.545,E2 8424.545} C_VEL
LIN {X 0,Y 595.308,Z 859.31,A -85,B 0,C 180,E1 8429.933,E2 8429.933} C_VEL
LIN {X 0,Y 595.438,Z 859.31,A -85,B 0,C 180,E1 8434.375,E2 8434.375} C_VEL
LIN {X 0,Y 595.453,Z 859.31,A -85,B 0,C 180,E1 8439.137,E2 8439.137} C_VEL
LIN {X 0,Y 595.503,Z 859.31,A -85,B 0,C 180,E1 8445.265,E2 8445.265} C_VEL
LIN {X 0,Y 595.766,Z 859.31,A -85,B 0,C 180,E1 8449.749,E2 8449.749} C_VEL
LIN {X 0,Y 595.942,Z 859.31,A -85,B 0,C 180,E1 8454.166,E2 8454.166} C_VEL
LIN {X 0,Y 596.035,Z 859.31,A -85,B 0,C 180,E1 8458.546,E2 8458.546} C_VEL
LIN {X 0,Y 596.024,Z 859.31,A -85,B 0,C 180,E1 8462.916,E2 8462.916} C_VEL
LIN {X 0,Y 595.803,Z 859.31,A -85,B 0,C 180,E1 8467.306,E2 8467.306} C_VEL
LIN {X 0,Y 595.711,Z 859.31,A -85,B 0,C 180,E1 8471.74,E2 8471.74} C_VEL
LIN {X 0,Y 595.635,Z 859.31,A -85,B 0,C 180,E1 8476.248,E2 8476.248} C_VEL
LIN {X 0,Y 595.561,Z 859.31,A -85,B 0,C 180,E1 8480.864,E2 8480.864} C_VEL
LIN {X 0,Y 595.443,Z 859.31,A -85,B 0,C 180,E1 8485.629,E2 8485.629} C_VEL
LIN {X 0,Y 595.32,Z 859.31,A -85,B 0,C 180,E1 8490.595,E2 8490.595} C_VEL
LIN {X 0,Y 595.222,Z 859.31,A -85,B 0,C 180,E1 8495.832,E2 8495.832} C_VEL
LIN {X 0,Y 595.081,Z 859.31,A -85,B 0,C 180,E1 8501.446,E2 8501.446} C_VEL
LIN {X 0,Y 595.101,Z 859.31,A -85,B 0,C 180,E1 8506.568,E2 8506.568} C_VEL
LIN {X 0,Y 595.324,Z 860.084,A -85,B 0,C 180,E1 8511.876,E2 8511.876} C_VEL
LIN {X 0,Y 609.481,Z 892.287,A -85,B 0,C 180,E1 8513.253,E2 8513.253} C_VEL
LIN {X 0,Y 612.354,Z 909.114,A -85,B 0,C 180,E1 8513.662,E2 8513.662} C_VEL
LIN {X 0,Y 612.06,Z 926.776,A -85,B 0,C 180,E1 8513.959,E2 8513.959} C_VEL
LIN {X 0,Y 609.606,Z 973.895,A -85,B 0,C 180,E1 8515.094,E2 8515.094} C_VEL
LIN {X 0,Y 606.5,Z 1019.763,A -85,B 0,C 180,E1 8516.845,E2 8516.845} C_VEL
LIN {X 0,Y 602.796,Z 1063.479,A -85,B 0,C 180,E1 8519.172,E2 8519.172} C_VEL
LIN {X 0,Y 598.983,Z 1103.513,A -85,B 0,C 180,E1 8522.035,E2 8522.035} C_VEL
LIN {X 0,Y 595.555,Z 1137.081,A -85,B 0,C 180,E1 8525.177,E2 8525.177} C_VEL
LIN {X 0,Y 592.862,Z 1164.844,A -85,B 0,C 180,E1 8528.499,E2 8528.499} C_VEL
LIN {X 0,Y 590.62,Z 1189.187,A -85,B 0,C 180,E1 8532.262,E2 8532.262} C_VEL
LIN {X 0,Y 589.274,Z 1208.067,A -85,B 0,C 180,E1 8536.24,E2 8536.24} C_VEL
LIN {X 0,Y 588.649,Z 1222.233,A -85,B 0,C 180,E1 8540.368,E2 8540.368} C_VEL
LIN {X 0,Y 588.434,Z 1231.667,A -85,B 0,C 180,E1 8544.829,E2 8544.829} C_VEL
LIN {X 0,Y 588.409,Z 1235.165,A -85,B 0,C 180,E1 8548.524,E2 8548.524} C_VEL
LIN {X 0,Y 588.372,Z 1234.213,A -85,B 0,C 180,E1 8552.952,E2 8552.952} C_VEL
LIN {X 0,Y 588.432,Z 1229.199,A -85,B 0,C 180,E1 8556.654,E2 8556.654} C_VEL
LIN {X 0,Y 588.8,Z 1217.72,A -85,B 0,C 180,E1 8561.129,E2 8561.129} C_VEL
LIN {X 0,Y 589.805,Z 1201.064,A -85,B 0,C 180,E1 8565.369,E2 8565.369} C_VEL
LIN {X 0,Y 591.465,Z 1180.701,A -85,B 0,C 180,E1 8569.175,E2 8569.175} C_VEL
LIN {X 0,Y 593.948,Z 1153.551,A -85,B 0,C 180,E1 8572.954,E2 8572.954} C_VEL
LIN {X 0,Y 597.249,Z 1120.694,A -85,B 0,C 180,E1 8576.46,E2 8576.46} C_VEL
LIN {X 0,Y 600.608,Z 1086.279,A -85,B 0,C 180,E1 8579.29,E2 8579.29} C_VEL
LIN {X 0,Y 604.207,Z 1047.159,A -85,B 0,C 180,E1 8581.78,E2 8581.78} C_VEL
LIN {X 0,Y 607.702,Z 1003.24,A -85,B 0,C 180,E1 8583.858,E2 8583.858} C_VEL
LIN {X 0,Y 610.676,Z 957.452,A -85,B 0,C 180,E1 8585.37,E2 8585.37} C_VEL
LIN {X 0,Y 611.781,Z 915.257,A -85,B 0,C 180,E1 8586.262,E2 8586.262} C_VEL
LIN {X 0,Y 588.894,Z 864.016,A -85,B 0,C 180,E1 8588.494,E2 8588.494} C_VEL
LIN {X 0,Y 587.319,Z 859.31,A -85,B 0,C 180,E1 8588.75,E2 8588.75} C_VEL
LIN {X 0,Y 587.367,Z 859.31,A -85,B 0,C 180,E1 8594.15,E2 8594.15} C_VEL
LIN {X 0,Y 587.245,Z 859.31,A -85,B 0,C 180,E1 8599.838,E2 8599.838} C_VEL
LIN {X 0,Y 587.271,Z 859.31,A -85,B 0,C 180,E1 8605.656,E2 8605.656} C_VEL
LIN {X 0,Y 587.448,Z 859.31,A -85,B 0,C 180,E1 8611.284,E2 8611.284} C_VEL
LIN {X 0,Y 587.553,Z 859.31,A -85,B 0,C 180,E1 8615.634,E2 8615.634} C_VEL
LIN {X 0,Y 587.67,Z 859.31,A -85,B 0,C 180,E1 8620.418,E2 8620.418} C_VEL
LIN {X 0,Y 587.705,Z 859.31,A -85,B 0,C 180,E1 8625.061,E2 8625.061} C_VEL
LIN {X 0,Y 587.814,Z 859.31,A -85,B 0,C 180,E1 8629.605,E2 8629.605} C_VEL
LIN {X 0,Y 588.015,Z 859.31,A -85,B 0,C 180,E1 8634.083,E2 8634.083} C_VEL
LIN {X 0,Y 588.146,Z 859.31,A -85,B 0,C 180,E1 8638.522,E2 8638.522} C_VEL
LIN {X 0,Y 588.119,Z 859.31,A -85,B 0,C 180,E1 8642.951,E2 8642.951} C_VEL
LIN {X 0,Y 587.934,Z 859.31,A -85,B 0,C 180,E1 8647.4,E2 8647.4} C_VEL
LIN {X 0,Y 587.761,Z 859.31,A -85,B 0,C 180,E1 8653.411,E2 8653.411} C_VEL
LIN {X 0,Y 587.695,Z 859.31,A -85,B 0,C 180,E1 8658.016,E2 8658.016} C_VEL
LIN {X 0,Y 587.559,Z 859.31,A -85,B 0,C 180,E1 8662.75,E2 8662.75} C_VEL
LIN {X 0,Y 587.406,Z 859.31,A -85,B 0,C 180,E1 8668.709,E2 8668.709} C_VEL
LIN {X 0,Y 587.287,Z 859.31,A -85,B 0,C 180,E1 8674.572,E2 8674.572} C_VEL
LIN {X 0,Y 587.226,Z 859.31,A -85,B 0,C 180,E1 8680.158,E2 8680.158} C_VEL
LIN {X 0,Y 587.193,Z 859.31,A -85,B 0,C 180,E1 8686.247,E2 8686.247} C_VEL
LIN {X 0,Y 587.261,Z 859.31,A -85,B 0,C 180,E1 8691.738,E2 8691.738} C_VEL
LIN {X 0,Y 587.342,Z 859.31,A -85,B 0,C 180,E1 8697.58,E2 8697.58} C_VEL
LIN {X 0,Y 610.679,Z 907.306,A -85,B 0,C 180,E1 8699.771,E2 8699.771} C_VEL
LIN {X 0,Y 609.686,Z 971.65,A -85,B 0,C 180,E1 8700.663,E2 8700.663} C_VEL
LIN {X 0,Y 607.321,Z 1011.018,A -85,B 0,C 180,E1 8701.762,E2 8701.762} C_VEL
LIN {X 0,Y 603.941,Z 1049.393,A -85,B 0,C 180,E1 8703.454,E2 8703.454} C_VEL
LIN {X 0,Y 600.138,Z 1084.417,A -85,B 0,C 180,E1 8705.656,E2 8705.656} C_VEL
LIN {X 0,Y 596.267,Z 1116.457,A -85,B 0,C 180,E1 8708.4,E2 8708.4} C_VEL
LIN {X 0,Y 593.167,Z 1142.959,A -85,B 0,C 180,E1 8711.432,E2 8711.432} C_VEL
LIN {X 0,Y 590.762,Z 1165.308,A -85,B 0,C 180,E1 8714.826,E2 8714.826} C_VEL
LIN {X 0,Y 589.328,Z 1183.202,A -85,B 0,C 180,E1 8718.506,E2 8718.506} C_VEL
LIN {X 0,Y 588.746,Z 1194.818,A -85,B 0,C 180,E1 8721.875,E2 8721.875} C_VEL
LIN {X 0,Y 588.415,Z 1202.759,A -85,B 0,C 180,E1 8725.569,E2 8725.569} C_VEL
LIN {X 0,Y 588.285,Z 1205.751,A -85,B 0,C 180,E1 8728.524,E2 8728.524} C_VEL
LIN {X 0,Y 588.388,Z 1205.687,A -85,B 0,C 180,E1 8731.476,E2 8731.476} C_VEL
LIN {X 0,Y 588.507,Z 1201.443,A -85,B 0,C 180,E1 8735.171,E2 8735.171} C_VEL
LIN {X 0,Y 588.809,Z 1191.129,A -85,B 0,C 180,E1 8739.256,E2 8739.256} C_VEL
LIN {X 0,Y 589.888,Z 1175.633,A -85,B 0,C 180,E1 8743.114,E2 8743.114} C_VEL
LIN {X 0,Y 591.909,Z 1153.933,A -85,B 0,C 180,E1 8746.93,E2 8746.93} C_VEL
LIN {X 0,Y 594.725,Z 1129.527,A -85,B 0,C 180,E1 8750.119,E2 8750.119} C_VEL
LIN {X 0,Y 598.264,Z 1100.026,A -85,B 0,C 180,E1 8753.017,E2 8753.017} C_VEL
LIN {X 0,Y 602.065,Z 1067.034,A -85,B 0,C 180,E1 8755.432,E2 8755.432} C_VEL
LIN {X 0,Y 605.602,Z 1031.796,A -85,B 0,C 180,E1 8757.308,E2 8757.308} C_VEL
LIN {X 0,Y 608.374,Z 994.349,A -85,B 0,C 180,E1 8758.684,E2 8758.684} C_VEL
LIN {X 0,Y 610.188,Z 954.834,A -85,B 0,C 180,E1 8759.546,E2 8759.546} C_VEL
LIN {X 0,Y 610.085,Z 906.056,A -85,B 0,C 180,E1 8760.189,E2 8760.189} C_VEL
LIN {X 0,Y 587.375,Z 859.31,A -85,B 0,C 180,E1 8762.366,E2 8762.366} C_VEL
LIN {X 0,Y 587.265,Z 859.31,A -85,B 0,C 180,E1 8768.262,E2 8768.262} C_VEL
LIN {X 0,Y 587.198,Z 859.31,A -85,B 0,C 180,E1 8774.167,E2 8774.167} C_VEL
LIN {X 0,Y 587.227,Z 859.31,A -85,B 0,C 180,E1 8779.842,E2 8779.842} C_VEL
LIN {X 0,Y 587.345,Z 859.31,A -85,B 0,C 180,E1 8785.647,E2 8785.647} C_VEL
LIN {X 0,Y 587.39,Z 859.31,A -85,B 0,C 180,E1 8791.295,E2 8791.295} C_VEL
LIN {X 0,Y 587.51,Z 859.31,A -85,B 0,C 180,E1 8795.637,E2 8795.637} C_VEL
LIN {X 0,Y 587.481,Z 859.31,A -85,B 0,C 180,E1 8800.416,E2 8800.416} C_VEL
LIN {X 0,Y 587.643,Z 859.31,A -85,B 0,C 180,E1 8806.587,E2 8806.587} C_VEL
LIN {X 0,Y 587.981,Z 859.31,A -85,B 0,C 180,E1 8812.156,E2 8812.156} C_VEL
LIN {X 0,Y 588.179,Z 859.31,A -85,B 0,C 180,E1 8817.049,E2 8817.049} C_VEL
LIN {X 0,Y 588.299,Z 859.31,A -85,B 0,C 180,E1 8821.478,E2 8821.478} C_VEL
LIN {X 0,Y 588.058,Z 859.31,A -85,B 0,C 180,E1 8825.916,E2 8825.916} C_VEL
LIN {X 0,Y 587.81,Z 859.31,A -85,B 0,C 180,E1 8831.9,E2 8831.9} C_VEL
